C05488=1204.604,-6.269,-42.765,-179.791,5.566,148.916
C05489=1204.600,-6.020,-42.779,-179.789,5.567,148.915
C05490=1204.595,-5.770,-42.793,-179.786,5.567,148.915
C05491=1204.589,-5.521,-42.806,-179.783,5.568,148.914
C05492=1204.584,-5.271,-42.821,-179.781,5.568,148.913
C05493=1204.580,-5.022,-42.834,-179.779,5.568,148.913
C05494=1204.574,-4.772,-42.848,-179.776,5.569,148.912
C05495=1204.569,-4.522,-42.862,-179.773,5.569,148.911
C05496=1204.564,-4.273,-42.876,-179.771,5.570,148.911
C05497=1204.560,-4.024,-42.889,-179.769,5.570,148.910
C05498=1204.554,-3.774,-42.903,-179.766,5.571,148.909
C05499=1204.549,-3.525,-42.917,-179.764,5.571,148.909
C05500=1204.544,-3.275,-42.931,-179.761,5.571,148.908
C05501=1204.539,-3.025,-42.946,-179.759,5.572,148.907
C05502=1204.535,-2.776,-42.959,-179.756,5.572,148.907
C05503=1204.529,-2.526,-42.972,-179.754,5.573,148.906
C05504=1204.524,-2.276,-42.987,-179.751,5.573,148.905
C05505=1204.519,-2.027,-43.001,-179.749,5.573,148.905
C05506=1204.513,-1.778,-43.015,-179.746,5.574,148.904
C05507=1204.508,-1.528,-43.029,-179.744,5.574,148.903
C05508=1204.504,-1.278,-43.042,-179.741,5.575,148.903
C05509=1204.498,-1.029,-43.056,-179.738,5.575,148.902
C05510=1204.493,-0.779,-43.070,-179.736,5.576,148.902
C05511=1204.488,-0.529,-43.085,-179.734,5.576,148.901
C05512=1204.483,-0.280,-43.099,-179.732,5.576,148.900
C05513=1204.478,-0.031,-43.113,-179.729,5.577,148.899
C05514=1204.473,0.219,-43.127,-179.726,5.577,148.899
C05515=1204.468,0.469,-43.140,-179.724,5.578,148.898
C05516=1204.463,0.718,-43.154,-179.721,5.578,148.898
C05517=1204.458,0.968,-43.168,-179.719,5.579,148.897
C05518=1204.453,1.217,-43.182,-179.716,5.579,148.896
C05519=1204.448,1.467,-43.197,-179.714,5.579,148.896
C05520=1204.442,1.716,-43.211,-179.711,5.580,148.895
C05521=1204.437,1.966,-43.225,-179.709,5.580,148.894
C05522=1204.433,2.216,-43.239,-179.706,5.581,148.894
C05523=1204.428,2.465,-43.253,-179.704,5.582,148.893
C05524=1204.422,2.735,-43.268,-179.701,5.582,148.892
C05525=1204.416,3.003,-43.284,-179.698,5.582,148.891
C05526=1204.411,3.272,-43.299,-179.695,5.583,148.891
C05527=1204.406,3.542,-43.314,-179.693,5.583,148.890
C05528=1204.401,3.791,-43.328,-179.690,5.584,148.889
C05529=1204.396,4.041,-43.342,-179.688,5.585,148.889
C05530=1204.390,4.290,-43.356,-179.686,5.584,148.888
C05531=1204.385,4.540,-43.371,-179.683,5.585,148.888
C05532=1204.380,4.789,-43.385,-179.681,5.585,148.887
C05533=1204.376,5.039,-43.400,-179.678,5.586,148.886
C05534=1204.371,5.288,-43.414,-179.675,5.586,148.886
C05535=1204.365,5.537,-43.428,-179.673,5.587,148.885
C05536=1204.360,5.787,-43.442,-179.670,5.588,148.884
C05537=1204.355,6.037,-43.457,-179.668,5.588,148.884
C05538=1204.350,6.286,-43.471,-179.666,5.588,148.883
C05539=1204.345,6.536,-43.485,-179.663,5.588,148.882
C05540=1204.340,6.786,-43.499,-179.660,5.589,148.882
C05541=1204.335,7.035,-43.513,-179.658,5.589,148.881
C05542=1204.330,7.285,-43.528,-179.656,5.590,148.880
C05543=1204.325,7.534,-43.542,-179.653,5.591,148.880
C05544=1204.320,7.784,-43.556,-179.650,5.591,148.879
C05545=1204.315,8.033,-43.571,-179.648,5.592,148.878
C05546=1204.310,8.283,-43.585,-179.645,5.592,148.878
C05547=1204.305,8.532,-43.599,-179.643,5.592,148.877
C05548=1204.300,8.781,-43.614,-179.641,5.593,148.877
C05549=1204.295,9.031,-43.628,-179.638,5.593,148.876
C05550=1204.290,9.281,-43.642,-179.635,5.594,148.875
C05551=1204.285,9.530,-43.657,-179.633,5.594,148.875
C05552=1204.279,9.780,-43.672,-179.630,5.595,148.874
C05553=1204.275,10.030,-43.686,-179.628,5.595,148.873
C05554=1204.270,10.279,-43.701,-179.625,5.596,148.872
C05555=1204.264,10.528,-43.714,-179.623,5.597,148.872
C05556=1204.259,10.778,-43.729,-179.620,5.597,148.871
C05557=1204.254,11.027,-43.744,-179.618,5.597,148.871
C05558=1204.249,11.277,-43.758,-179.615,5.597,148.870
C05559=1204.244,11.527,-43.772,-179.613,5.598,148.869
C05560=1204.239,11.776,-43.788,-179.610,5.598,148.869
C05561=1204.234,12.026,-43.802,-179.608,5.599,148.868
C05562=1204.229,12.275,-43.816,-179.605,5.600,148.867
C05563=1204.224,12.525,-43.831,-179.603,5.600,148.867
C05564=1204.219,12.774,-43.845,-179.600,5.601,148.866
C05565=1204.214,13.023,-43.860,-179.597,5.601,148.865
C05566=1204.209,13.273,-43.874,-179.595,5.602,148.865
C05567=1204.204,13.522,-43.889,-179.593,5.602,148.864
C05568=1204.199,13.772,-43.904,-179.590,5.602,148.864
C05569=1204.194,14.022,-43.918,-179.588,5.603,148.863
C05570=1204.189,14.271,-43.933,-179.585,5.603,148.862
C05571=1204.184,14.521,-43.947,-179.582,5.604,148.862
C05572=1204.178,14.771,-43.962,-179.580,5.604,148.861
C05573=1204.174,15.020,-43.977,-179.578,5.605,148.860
C05574=1204.169,15.269,-43.991,-179.575,5.606,148.860
C05575=1204.164,15.519,-44.006,-179.572,5.606,148.859
C05576=1204.159,15.769,-44.021,-179.570,5.607,148.858
C05577=1204.154,16.018,-44.036,-179.567,5.607,148.858
C05578=1204.149,16.267,-44.051,-179.565,5.608,148.857
C05579=1204.144,16.517,-44.065,-179.562,5.609,148.857
C05580=1204.138,16.767,-44.080,-179.560,5.608,148.856
C05581=1204.134,17.016,-44.095,-179.558,5.609,148.855
C05582=1204.129,17.266,-44.109,-179.555,5.609,148.854
C05583=1204.124,17.515,-44.124,-179.552,5.610,148.854
C05584=1204.118,17.765,-44.139,-179.550,5.611,148.853
C05585=1204.114,18.014,-44.154,-179.547,5.611,148.853
C05586=1204.109,18.264,-44.168,-179.545,5.612,148.852
C05587=1204.104,18.514,-44.182,-179.542,5.612,148.851
C05588=1204.098,18.763,-44.198,-179.539,5.613,148.851
C05589=1204.093,19.013,-44.212,-179.537,5.613,148.850
C05590=1204.089,19.262,-44.227,-179.535,5.614,148.849
C05591=1204.083,19.512,-44.242,-179.532,5.615,148.849
C05592=1204.078,19.761,-44.257,-179.529,5.615,148.848
C05593=1204.074,20.010,-44.272,-179.527,5.616,148.847
C05594=1204.068,20.260,-44.287,-179.524,5.616,148.847
C05595=1204.063,20.509,-44.302,-179.522,5.617,148.846
C05596=1204.059,20.759,-44.316,-179.520,5.617,148.846
C05597=1204.053,21.008,-44.332,-179.517,5.617,148.845
C05598=1204.048,21.258,-44.346,-179.515,5.618,148.844
C05599=1204.044,21.507,-44.361,-179.512,5.618,148.844
C05600=1204.038,21.757,-44.376,-179.509,5.619,148.843
C05601=1204.033,22.006,-44.391,-179.507,5.620,148.842
C05602=1204.028,22.255,-44.407,-179.504,5.620,148.842
C05603=1204.023,22.505,-44.421,-179.502,5.621,148.841
C05604=1204.018,22.754,-44.436,-179.499,5.621,148.840
C05605=1204.012,23.004,-44.451,-179.497,5.622,148.840
C05606=1204.008,23.253,-44.466,-179.494,5.623,148.839
C05607=1204.002,23.503,-44.481,-179.492,5.623,148.839
C05608=1203.998,23.753,-44.496,-179.489,5.624,148.838
C05609=1203.993,24.002,-44.511,-179.486,5.624,148.837
C05610=1203.988,24.252,-44.527,-179.484,5.625,148.837
C05611=1203.983,24.501,-44.541,-179.482,5.626,148.836
C05612=1203.978,24.751,-44.556,-179.479,5.626,148.835
C05613=1203.973,25.000,-44.571,-179.476,5.627,148.835
C05614=1203.967,25.250,-44.586,-179.474,5.627,148.834
C05615=1203.963,25.499,-44.601,-179.471,5.628,148.833
C05616=1203.957,25.748,-44.617,-179.468,5.628,148.833
C05617=1203.953,25.998,-44.632,-179.466,5.629,148.832
C05618=1203.948,26.248,-44.646,-179.464,5.630,148.832
C05619=1203.943,26.497,-44.662,-179.461,5.630,148.831
C05620=1203.938,26.746,-44.677,-179.458,5.631,148.830
C05621=1203.933,26.996,-44.693,-179.456,5.631,148.830
C05622=1203.928,27.246,-44.707,-179.453,5.632,148.829
C05623=1203.923,27.495,-44.723,-179.451,5.632,148.828
C05624=1203.918,27.744,-44.738,-179.449,5.632,148.828
C05625=1203.913,27.994,-44.753,-179.446,5.633,148.827
C05626=1203.907,28.244,-44.768,-179.443,5.633,148.826
C05627=1203.903,28.493,-44.783,-179.441,5.634,148.826
C05628=1203.897,28.762,-44.800,-179.438,5.636,148.825
C05629=1203.892,29.030,-44.816,-179.435,5.636,148.825
C05630=1203.887,29.299,-44.833,-179.433,5.637,148.824
C05631=1203.881,29.568,-44.849,-179.430,5.637,148.823
C05632=1203.876,29.817,-44.864,-179.428,5.638,148.823
C05633=1203.871,30.067,-44.880,-179.425,5.638,148.822
C05634=1203.867,30.316,-44.895,-179.422,5.639,148.821
C05635=1203.861,30.566,-44.911,-179.420,5.639,148.820
C05636=1203.856,30.815,-44.925,-179.417,5.640,148.820
C05637=1203.851,31.065,-44.941,-179.415,5.641,148.819
C05638=1203.846,31.314,-44.956,-179.412,5.641,148.819
C05639=1203.841,31.564,-44.972,-179.410,5.642,148.818
C05640=1203.836,31.813,-44.987,-179.407,5.642,148.817
C05641=1203.831,32.063,-45.002,-179.405,5.643,148.817
C05642=1203.826,32.312,-45.018,-179.402,5.644,148.816
C05643=1203.821,32.562,-45.034,-179.399,5.644,148.816
C05644=1203.817,32.811,-45.049,-179.397,5.645,148.815
C05645=1203.811,33.061,-45.064,-179.395,5.646,148.814
C05646=1203.807,33.310,-45.079,-179.392,5.646,148.814
C05647=1203.801,33.559,-45.095,-179.389,5.647,148.813
C05648=1203.796,33.809,-45.111,-179.387,5.647,148.812
C05649=1203.792,34.058,-45.126,-179.384,5.648,148.812
C05650=1203.786,34.308,-45.142,-179.382,5.649,148.811
C05651=1203.781,34.557,-45.157,-179.379,5.649,148.811
C05652=1203.777,34.807,-45.172,-179.377,5.650,148.810
C05653=1203.772,35.056,-45.188,-179.374,5.650,148.809
C05654=1203.766,35.306,-45.204,-179.371,5.651,148.809
C05655=1203.761,35.555,-45.219,-179.369,5.652,148.808
C05656=1203.757,35.805,-45.235,-179.367,5.652,148.807
C05657=1203.751,36.054,-45.250,-179.364,5.653,148.807
C05658=1203.746,36.304,-45.266,-179.361,5.653,148.806
C05659=1203.742,36.553,-45.281,-179.359,5.654,148.806
C05660=1203.736,36.803,-45.297,-179.356,5.655,148.805
C05661=1203.731,37.052,-45.312,-179.354,5.655,148.804
C05662=1203.726,37.302,-45.328,-179.351,5.656,148.804
C05663=1203.722,37.551,-45.344,-179.349,5.656,148.803
C05664=1203.717,37.800,-45.360,-179.346,5.657,148.802
C05665=1203.711,38.050,-45.375,-179.344,5.658,148.802
C05666=1203.706,38.300,-45.391,-179.341,5.658,148.801
C05667=1203.702,38.549,-45.406,-179.338,5.659,148.800
C05668=1203.696,38.798,-45.422,-179.336,5.660,148.800
C05669=1203.692,39.048,-45.438,-179.334,5.660,148.799
C05670=1203.687,39.297,-45.454,-179.330,5.661,148.799
C05671=1203.681,39.547,-45.470,-179.328,5.662,148.798
C05672=1203.677,39.796,-45.485,-179.325,5.663,148.797
C05673=1203.672,40.046,-45.500,-179.323,5.663,148.797
C05674=1203.666,40.295,-45.516,-179.320,5.664,148.796
C05675=1203.662,40.545,-45.533,-179.318,5.664,148.796
C05676=1203.656,40.794,-45.548,-179.315,5.665,148.795
C05677=1203.652,41.043,-45.563,-179.313,5.666,148.794
C05678=1203.647,41.293,-45.579,-179.310,5.666,148.794
C05679=1203.642,41.543,-45.595,-179.308,5.667,148.793
C05680=1203.637,41.791,-45.611,-179.305,5.668,148.792
C05681=1203.632,42.041,-45.627,-179.303,5.668,148.792
C05682=1203.626,42.291,-45.643,-179.300,5.669,148.791
C05683=1203.621,42.540,-45.659,-179.298,5.669,148.791
C05684=1203.617,42.789,-45.674,-179.295,5.670,148.790
C05685=1203.612,43.039,-45.690,-179.293,5.671,148.789
C05686=1203.607,43.289,-45.706,-179.290,5.671,148.789
C05687=1203.602,43.538,-45.722,-179.288,5.672,148.788
C05688=1203.597,43.787,-45.738,-179.285,5.673,148.787
C05689=1203.592,44.037,-45.754,-179.283,5.673,148.787
C05690=1203.587,44.286,-45.770,-179.280,5.675,148.786
C05691=1203.582,44.536,-45.786,-179.277,5.675,148.786
C05692=1203.577,44.786,-45.802,-179.274,5.676,148.785
C05693=1203.572,45.034,-45.817,-179.272,5.677,148.785
C05694=1203.567,45.284,-45.833,-179.269,5.677,148.784
C05695=1203.562,45.533,-45.850,-179.267,5.678,148.783
C05696=1203.558,45.783,-45.866,-179.264,5.678,148.783
C05697=1203.552,46.032,-45.881,-179.262,5.679,148.782
C05698=1203.548,46.282,-45.898,-179.259,5.680,148.781
C05699=1203.542,46.531,-45.913,-179.257,5.680,148.781
C05700=1203.537,46.780,-45.930,-179.254,5.681,148.780
C05701=1203.532,47.030,-45.946,-179.252,5.682,148.780
C05702=1203.527,47.279,-45.962,-179.249,5.682,148.779
C05703=1203.523,47.529,-45.978,-179.246,5.684,148.778
C05704=1203.517,47.778,-45.993,-179.243,5.684,148.778
C05705=1203.513,48.028,-46.010,-179.241,5.685,148.777
C05706=1203.507,48.277,-46.026,-179.239,5.686,148.777
C05707=1203.503,48.527,-46.042,-179.236,5.686,148.776
C05708=1203.497,48.776,-46.058,-179.233,5.687,148.775
C05709=1203.493,49.026,-46.075,-179.231,5.688,148.775
C05710=1203.488,49.275,-46.090,-179.229,5.688,148.774
C05711=1203.483,49.525,-46.107,-179.226,5.689,148.773
C05712=1203.478,49.773,-46.123,-179.223,5.689,148.773
C05713=1203.473,50.024,-46.139,-179.221,5.690,148.772
C05714=1203.468,50.272,-46.155,-179.219,5.691,148.772
C05715=1203.463,50.522,-46.171,-179.215,5.692,148.771
C05716=1203.458,50.771,-46.188,-179.213,5.693,148.770
C05717=1203.454,51.021,-46.204,-179.211,5.693,148.770
C05718=1203.448,51.270,-46.220,-179.208,5.694,148.769
C05719=1203.443,51.520,-46.237,-179.205,5.694,148.769
C05720=1203.438,51.769,-46.253,-179.203,5.695,148.768
C05721=1203.433,52.019,-46.269,-179.200,5.696,148.767
C05722=1203.428,52.268,-46.285,-179.198,5.696,148.767
C05723=1203.423,52.518,-46.302,-179.195,5.697,148.766
C05724=1203.418,52.766,-46.318,-179.193,5.698,148.766
C05725=1203.414,53.017,-46.334,-179.190,5.699,148.765
C05726=1203.409,53.265,-46.350,-179.187,5.700,148.764
C05727=1203.404,53.515,-46.367,-179.185,5.700,148.764
C05728=1203.399,53.764,-46.383,-179.182,5.701,148.763
C05729=1203.393,54.014,-46.400,-179.180,5.702,148.763
C05730=1203.389,54.263,-46.417,-179.177,5.702,148.762
C05731=1203.384,54.513,-46.432,-179.175,5.703,148.761
C05732=1203.379,54.781,-46.450,-179.172,5.705,148.761
C05733=1203.373,55.050,-46.467,-179.169,5.705,148.760
C05734=1203.367,55.318,-46.486,-179.167,5.706,148.759
C05735=1203.362,55.587,-46.503,-179.164,5.706,148.759
C05736=1203.357,55.836,-46.519,-179.161,5.708,148.758
C05737=1203.353,56.086,-46.536,-179.158,5.708,148.757
C05738=1203.348,56.334,-46.552,-179.156,5.709,148.757
C05739=1203.342,56.585,-46.569,-179.153,5.710,148.756
C05740=1203.338,56.834,-46.585,-179.151,5.710,148.756
C05741=1203.333,57.083,-46.602,-179.148,5.711,148.755
C05742=1203.328,57.332,-46.618,-179.146,5.712,148.755
C05743=1203.322,57.582,-46.635,-179.143,5.712,148.754
C05744=1203.318,57.832,-46.651,-179.140,5.713,148.753
C05745=1203.313,58.081,-46.668,-179.138,5.714,148.753
C05746=1203.308,58.330,-46.684,-179.135,5.715,148.752
C05747=1203.304,58.579,-46.701,-179.133,5.715,148.751
C05748=1203.298,58.829,-46.718,-179.130,5.716,148.751
C05749=1203.293,59.078,-46.734,-179.128,5.717,148.750
C05750=1203.289,59.327,-46.751,-179.125,5.717,148.750
C05751=1203.283,59.577,-46.767,-179.122,5.719,148.749
C05752=1203.278,59.827,-46.784,-179.120,5.720,148.749
C05753=1203.274,60.076,-46.801,-179.117,5.720,148.748
C05754=1203.269,60.325,-46.817,-179.115,5.721,148.747
C05755=1203.263,60.575,-46.834,-179.112,5.722,148.747
C05756=1203.259,60.824,-46.851,-179.110,5.722,148.746
C05757=1203.254,61.073,-46.867,-179.107,5.723,148.746
C05758=1203.249,61.323,-46.884,-179.104,5.725,148.745
C05759=1203.244,61.572,-46.901,-179.102,5.725,148.744
C05760=1203.239,61.821,-46.917,-179.099,5.726,148.744
C05761=1203.234,62.071,-46.935,-179.097,5.726,148.743
C05762=1203.229,62.320,-46.951,-179.094,5.727,148.743
C05763=1203.225,62.570,-46.968,-179.092,5.728,148.742
C05764=1203.219,62.819,-46.985,-179.089,5.729,148.741
C05765=1203.215,63.068,-47.002,-179.086,5.730,148.741
C05766=1203.210,63.318,-47.018,-179.084,5.730,148.740
C05767=1203.204,63.567,-47.035,-179.081,5.731,148.740
C05768=1203.200,63.816,-47.052,-179.079,5.732,148.739
C05769=1203.195,64.066,-47.069,-179.076,5.732,148.738
C05770=1203.190,64.316,-47.086,-179.073,5.734,148.738
C05771=1203.185,64.565,-47.102,-179.071,5.735,148.737
C05772=1203.180,64.814,-47.119,-179.068,5.735,148.737
C05773=1203.175,65.064,-47.136,-179.066,5.736,148.736
C05774=1203.170,65.313,-47.153,-179.064,5.737,148.736
C05775=1203.165,65.562,-47.170,-179.061,5.737,148.735
C05776=1203.161,65.812,-47.186,-179.058,5.739,148.734
C05777=1203.155,66.062,-47.203,-179.056,5.740,148.734
C05778=1203.150,66.310,-47.220,-179.053,5.740,148.733
C05779=1203.145,66.560,-47.238,-179.050,5.741,148.733
C05780=1203.141,66.809,-47.254,-179.048,5.741,148.732
C05781=1203.136,67.059,-47.272,-179.045,5.743,148.731
C05782=1203.131,67.308,-47.288,-179.042,5.744,148.731
C05783=1203.125,67.557,-47.305,-179.040,5.744,148.730
C05784=1203.121,67.807,-47.322,-179.038,5.745,148.730
C05785=1203.116,68.057,-47.339,-179.035,5.746,148.729
C05786=1203.111,68.306,-47.357,-179.032,5.746,148.728
C05787=1203.106,68.555,-47.373,-179.030,5.748,148.728
C05788=1203.101,68.804,-47.390,-179.027,5.748,148.727
C05789=1203.096,69.054,-47.407,-179.024,5.749,148.727
C05790=1203.092,69.303,-47.425,-179.022,5.750,148.726
C05791=1203.087,69.553,-47.442,-179.020,5.750,148.726
C05792=1203.081,69.801,-47.458,-179.016,5.752,148.725
C05793=1203.076,70.051,-47.476,-179.014,5.753,148.724
C05794=1203.072,70.300,-47.493,-179.012,5.753,148.724
C05795=1203.067,70.550,-47.510,-179.009,5.754,148.723
C05796=1203.062,70.799,-47.527,-179.007,5.755,148.723
C05797=1203.057,71.049,-47.544,-179.004,5.756,148.722
C05798=1203.052,71.297,-47.561,-179.001,5.757,148.721
C05799=1203.047,71.547,-47.579,-178.999,5.758,148.721
C05800=1203.042,71.797,-47.596,-178.996,5.758,148.720
C05801=1203.038,72.046,-47.613,-178.994,5.760,148.720
C05802=1203.033,72.296,-47.630,-178.991,5.760,148.719
C05803=1203.028,72.545,-47.647,-178.988,5.761,148.719
C05804=1203.023,72.794,-47.665,-178.986,5.762,148.718
C05805=1203.017,73.043,-47.682,-178.984,5.762,148.717
C05806=1203.013,73.293,-47.699,-178.980,5.764,148.717
C05807=1203.008,73.542,-47.717,-178.978,5.765,148.716
C05808=1203.003,73.791,-47.733,-178.976,5.765,148.716
C05809=1202.998,74.041,-47.751,-178.973,5.766,148.715
C05810=1202.993,74.290,-47.769,-178.971,5.767,148.715
C05811=1202.989,74.540,-47.785,-178.968,5.768,148.714
C05812=1202.984,74.789,-47.803,-178.965,5.769,148.713
C05813=1202.978,75.038,-47.820,-178.963,5.770,148.713
C05814=1202.974,75.287,-47.837,-178.960,5.770,148.712
C05815=1202.969,75.537,-47.855,-178.957,5.772,148.712
C05816=1202.964,75.786,-47.873,-178.955,5.772,148.711
C05817=1202.959,76.036,-47.889,-178.952,5.773,148.710
C05818=1202.954,76.285,-47.907,-178.950,5.774,148.710
C05819=1202.949,76.535,-47.925,-178.947,5.775,148.709
C05820=1202.944,76.784,-47.942,-178.944,5.776,148.709
C05821=1202.940,77.033,-47.959,-178.942,5.777,148.708
C05822=1202.935,77.283,-47.977,-178.939,5.777,148.708
C05823=1202.930,77.532,-47.995,-178.936,5.779,148.707
C05824=1202.925,77.782,-48.011,-178.934,5.780,148.707
C05825=1202.920,78.031,-48.029,-178.931,5.780,148.706
C05826=1202.915,78.279,-48.047,-178.929,5.781,148.705
C05827=1202.910,78.529,-48.064,-178.926,5.783,148.705
C05828=1202.905,78.778,-48.081,-178.924,5.783,148.704
C05829=1202.900,79.028,-48.099,-178.921,5.784,148.704
C05830=1202.895,79.277,-48.117,-178.919,5.785,148.703
C05831=1202.890,79.527,-48.134,-178.916,5.786,148.702
C05832=1202.885,79.776,-48.152,-178.913,5.787,148.702
C05833=1202.881,80.025,-48.169,-178.911,5.787,148.701
C05834=1202.876,80.275,-48.187,-178.909,5.788,148.701
C05835=1202.871,80.524,-48.205,-178.905,5.790,148.700
C05836=1202.865,80.793,-48.223,-178.903,5.790,148.700
C05837=1202.860,81.061,-48.243,-178.900,5.791,148.699
C05838=1202.855,81.329,-48.262,-178.897,5.792,148.698
C05839=1202.849,81.597,-48.280,-178.895,5.793,148.698
C05840=1202.845,81.846,-48.298,-178.892,5.795,148.697
C05841=1202.840,82.096,-48.315,-178.889,5.795,148.697
C05842=1202.836,82.346,-48.333,-178.887,5.796,148.696
C05843=1202.831,82.595,-48.351,-178.884,5.797,148.696
C05844=1202.826,82.844,-48.369,-178.882,5.798,148.695
C05845=1202.821,83.094,-48.387,-178.879,5.799,148.694
C05846=1202.816,83.343,-48.405,-178.876,5.799,148.694
C05847=1202.811,83.592,-48.422,-178.874,5.801,148.693
C05848=1202.807,83.841,-48.440,-178.871,5.802,148.693
C05849=1202.801,84.091,-48.457,-178.869,5.803,148.692
C05850=1202.796,84.340,-48.475,-178.866,5.803,148.692
C05851=1202.792,84.589,-48.493,-178.863,5.805,148.691
C05852=1202.787,84.838,-48.511,-178.861,5.806,148.691
C05853=1202.781,85.088,-48.528,-178.858,5.806,148.690
C05854=1202.776,85.337,-48.546,-178.856,5.807,148.690
C05855=1202.772,85.587,-48.564,-178.853,5.808,148.689
C05856=1202.767,85.836,-48.582,-178.850,5.809,148.688
C05857=1202.762,86.085,-48.600,-178.848,5.810,148.688
C05858=1202.757,86.334,-48.618,-178.845,5.811,148.687
C05859=1202.752,86.584,-48.635,-178.843,5.812,148.687
C05860=1202.748,86.834,-48.653,-178.840,5.813,148.686
C05861=1202.743,87.083,-48.671,-178.837,5.814,148.685
C05862=1202.738,87.332,-48.689,-178.835,5.815,148.685
C05863=1202.733,87.581,-48.707,-178.832,5.816,148.684
C05864=1202.728,87.830,-48.725,-178.830,5.817,148.684
C05865=1202.723,88.079,-48.743,-178.827,5.818,148.683
C05866=1202.719,88.329,-48.761,-178.824,5.819,148.683
C05867=1202.714,88.578,-48.779,-178.822,5.820,148.682
C05868=1202.709,88.827,-48.797,-178.819,5.821,148.682
C05869=1202.704,89.076,-48.815,-178.817,5.822,148.681
C05870=1202.699,89.327,-48.833,-178.814,5.822,148.680
C05871=1202.694,89.576,-48.851,-178.812,5.824,148.680
C05872=1202.689,89.825,-48.869,-178.809,5.825,148.679
C05873=1202.684,90.074,-48.887,-178.806,5.825,148.679
C05874=1202.679,90.324,-48.905,-178.804,5.827,148.678
C05875=1202.674,90.573,-48.923,-178.801,5.828,148.678
C05876=1202.669,90.822,-48.941,-178.799,5.829,148.677
C05877=1202.665,91.072,-48.960,-178.796,5.830,148.677
C05878=1202.660,91.321,-48.978,-178.793,5.831,148.676
C05879=1202.655,91.570,-48.996,-178.791,5.831,148.676
C05880=1202.650,91.819,-49.014,-178.788,5.833,148.675
C05881=1202.645,92.068,-49.032,-178.786,5.834,148.675
C05882=1202.641,92.318,-49.051,-178.783,5.834,148.674
C05883=1202.636,92.567,-49.069,-178.781,5.835,148.673
C05884=1202.631,92.816,-49.087,-178.778,5.837,148.673
C05885=1202.626,93.066,-49.105,-178.775,5.838,148.672
C05886=1202.621,93.315,-49.123,-178.773,5.838,148.672
C05887=1202.616,93.565,-49.141,-178.770,5.840,148.671
C05888=1202.611,93.814,-49.159,-178.768,5.840,148.671
C05889=1202.607,94.063,-49.177,-178.764,5.842,148.670
C05890=1202.602,94.312,-49.196,-178.762,5.843,148.670
C05891=1202.597,94.561,-49.214,-178.760,5.843,148.669
C05892=1202.592,94.811,-49.233,-178.757,5.845,148.669
C05893=1202.587,95.060,-49.251,-178.754,5.846,148.668
C05894=1202.582,95.309,-49.269,-178.752,5.847,148.667
C05895=1202.577,95.558,-49.287,-178.749,5.848,148.667
C05896=1202.573,95.807,-49.306,-178.747,5.849,148.666
C05897=1202.568,96.057,-49.325,-178.744,5.850,148.666
C05898=1202.563,96.306,-49.343,-178.741,5.851,148.665
C05899=1202.558,96.556,-49.361,-178.739,5.852,148.665
C05900=1202.553,96.805,-49.379,-178.736,5.852,148.664
C05901=1202.549,97.054,-49.398,-178.734,5.854,148.664
C05902=1202.543,97.304,-49.416,-178.731,5.855,148.663
C05903=1202.538,97.553,-49.434,-178.729,5.856,148.663
C05904=1202.534,97.802,-49.453,-178.726,5.857,148.662
C05905=1202.529,98.051,-49.471,-178.723,5.858,148.662
C05906=1202.524,98.301,-49.490,-178.721,5.859,148.661
C05907=1202.519,98.550,-49.508,-178.718,5.860,148.660
C05908=1202.515,98.799,-49.527,-178.716,5.861,148.660
C05909=1202.510,99.048,-49.545,-178.713,5.863,148.659
C05910=1202.504,99.298,-49.563,-178.710,5.863,148.659
C05911=1202.500,99.547,-49.582,-178.708,5.864,148.658
C05912=1202.495,99.796,-49.600,-178.705,5.866,148.658
C05913=1202.490,100.046,-49.619,-178.702,5.866,148.657
C05914=1202.486,100.295,-49.638,-178.700,5.867,148.657
C05915=1202.481,100.544,-49.656,-178.697,5.868,148.656
C05916=1202.475,100.793,-49.675,-178.695,5.869,148.656
C05917=1202.470,101.042,-49.693,-178.692,5.871,148.655
C05918=1202.466,101.292,-49.712,-178.689,5.872,148.655
C05919=1202.461,101.541,-49.731,-178.687,5.872,148.654
C05920=1202.456,101.790,-49.749,-178.684,5.874,148.653
C05921=1202.452,102.039,-49.768,-178.682,5.875,148.653
C05922=1202.446,102.289,-49.787,-178.679,5.876,148.652
C05923=1202.442,102.538,-49.806,-178.676,5.877,148.652
C05924=1202.437,102.787,-49.824,-178.674,5.878,148.651
C05925=1202.432,103.037,-49.842,-178.671,5.879,148.651
C05926=1202.428,103.286,-49.861,-178.669,5.880,148.650
C05927=1202.422,103.535,-49.880,-178.666,5.881,148.650
C05928=1202.417,103.784,-49.898,-178.663,5.883,148.649
C05929=1202.413,104.034,-49.917,-178.661,5.883,148.649
C05930=1202.408,104.283,-49.936,-178.658,5.885,148.648
C05931=1202.403,104.532,-49.954,-178.656,5.886,148.648
C05932=1202.398,104.781,-49.974,-178.653,5.886,148.647
C05933=1202.394,105.030,-49.992,-178.650,5.888,148.647
C05934=1202.388,105.280,-50.011,-178.648,5.889,148.646
C05935=1202.384,105.529,-50.030,-178.645,5.890,148.645
C05936=1202.379,105.778,-50.048,-178.643,5.891,148.645
C05937=1202.374,106.028,-50.068,-178.640,5.893,148.644
C05938=1202.369,106.277,-50.086,-178.637,5.893,148.644
C05939=1202.365,106.526,-50.105,-178.635,5.894,148.643
C05940=1202.359,106.794,-50.126,-178.632,5.895,148.643
C05941=1202.354,107.062,-50.145,-178.629,5.897,148.642
C05942=1202.349,107.331,-50.167,-178.626,5.898,148.642
C05943=1202.343,107.600,-50.187,-178.623,5.899,148.641
C05944=1202.339,107.849,-50.206,-178.621,5.900,148.641
C05945=1202.334,108.098,-50.224,-178.618,5.902,148.640
C05946=1202.330,108.348,-50.243,-178.616,5.903,148.640
C05947=1202.324,108.597,-50.263,-178.614,5.903,148.639
C05948=1202.320,108.846,-50.282,-178.610,5.905,148.639
C05949=1202.315,109.095,-50.300,-178.608,5.906,148.638
C05950=1202.310,109.344,-50.319,-178.605,5.907,148.638
C05951=1202.305,109.593,-50.339,-178.603,5.908,148.637
C05952=1202.300,109.843,-50.357,-178.600,5.910,148.636
C05953=1202.296,110.092,-50.376,-178.598,5.910,148.636
C05954=1202.290,110.341,-50.395,-178.594,5.912,148.635
C05955=1202.286,110.590,-50.415,-178.592,5.913,148.635
C05956=1202.281,110.840,-50.433,-178.590,5.913,148.634
C05957=1202.277,111.089,-50.452,-178.587,5.915,148.634
C05958=1202.271,111.338,-50.471,-178.584,5.916,148.633
C05959=1202.267,111.587,-50.491,-178.582,5.918,148.633
C05960=1202.262,111.836,-50.510,-178.579,5.918,148.632
C05961=1202.257,112.086,-50.529,-178.576,5.920,148.632
C05962=1202.252,112.335,-50.547,-178.574,5.920,148.631
C05963=1202.247,112.584,-50.567,-178.571,5.922,148.631
C05964=1202.242,112.833,-50.586,-178.569,5.923,148.630
C05965=1202.238,113.082,-50.605,-178.566,5.924,148.630
C05966=1202.233,113.332,-50.625,-178.564,5.926,148.629
C05967=1202.228,113.581,-50.644,-178.561,5.926,148.629
C05968=1202.224,113.831,-50.663,-178.558,5.928,148.628
C05969=1202.218,114.080,-50.682,-178.556,5.928,148.628
C05970=1202.214,114.329,-50.702,-178.553,5.930,148.627
C05971=1202.209,114.578,-50.720,-178.550,5.931,148.627
C05972=1202.204,114.827,-50.740,-178.548,5.933,148.626
C05973=1202.199,115.076,-50.759,-178.545,5.933,148.626
C05974=1202.195,115.325,-50.778,-178.542,5.935,148.625
C05975=1202.190,115.574,-50.798,-178.540,5.936,148.625
C05976=1202.185,115.824,-50.817,-178.537,5.937,148.624
C05977=1202.180,116.073,-50.837,-178.535,5.938,148.624
C05978=1202.175,116.322,-50.856,-178.532,5.939,148.623
C05979=1202.171,116.572,-50.875,-178.530,5.941,148.623
C05980=1202.165,116.820,-50.895,-178.527,5.941,148.622
C05981=1202.161,117.070,-50.914,-178.524,5.943,148.622
C05982=1202.157,117.319,-50.933,-178.522,5.944,148.621
C05983=1202.151,117.568,-50.953,-178.519,5.945,148.621
C05984=1202.147,117.818,-50.972,-178.517,5.946,148.620
C05985=1202.141,118.067,-50.992,-178.514,5.948,148.620
C05986=1202.136,118.316,-51.011,-178.512,5.949,148.619
C05987=1202.132,118.565,-51.030,-178.508,5.950,148.619
C05988=1202.127,118.814,-51.050,-178.506,5.951,148.618
C05989=1202.122,119.064,-51.069,-178.503,5.952,148.618
C05990=1202.118,119.313,-51.089,-178.501,5.953,148.617
C05991=1202.112,119.562,-51.108,-178.498,5.955,148.617
C05992=1202.109,119.811,-51.128,-178.496,5.956,148.616
C05993=1202.103,120.060,-51.147,-178.493,5.957,148.616
C05994=1202.099,120.309,-51.167,-178.490,5.958,148.615
C05995=1202.094,120.559,-51.187,-178.488,5.960,148.615
C05996=1202.088,120.808,-51.206,-178.486,5.961,148.614
C05997=1202.084,121.057,-51.226,-178.482,5.962,148.614
C05998=1202.079,121.306,-51.246,-178.480,5.963,148.613
C05999=1202.075,121.555,-51.265,-178.477,5.965,148.613
C06000=1202.070,121.804,-51.284,-178.475,5.965,148.612
C06001=1202.065,122.054,-51.304,-178.472,5.967,148.612
C06002=1202.060,122.304,-51.324,-178.470,5.968,148.611
C06003=1202.055,122.552,-51.344,-178.467,5.970,148.611
C06004=1202.051,122.801,-51.363,-178.464,5.970,148.610
C06005=1202.046,123.051,-51.383,-178.462,5.972,148.610
C06006=1202.041,123.300,-51.402,-178.459,5.973,148.609
C06007=1202.036,123.549,-51.423,-178.456,5.974,148.609
C06008=1202.031,123.798,-51.442,-178.454,5.975,148.608
C06009=1202.026,124.047,-51.462,-178.451,5.977,148.608
C06010=1202.022,124.296,-51.481,-178.449,5.978,148.607
C06011=1202.018,124.545,-51.501,-178.446,5.979,148.607
C06012=1202.013,124.795,-51.521,-178.444,5.980,148.606
C06013=1202.007,125.044,-51.540,-178.441,5.982,148.606
C06014=1202.003,125.293,-51.560,-178.438,5.983,148.605
C06015=1201.998,125.542,-51.580,-178.436,5.984,148.605
C06016=1201.994,125.792,-51.600,-178.433,5.986,148.604
C06017=1201.989,126.040,-51.620,-178.430,5.987,148.604
C06018=1201.984,126.290,-51.639,-178.428,5.988,148.603
C06019=1201.979,126.539,-51.660,-178.425,5.989,148.603
C06020=1201.975,126.788,-51.679,-178.422,5.991,148.602
C06021=1201.969,127.037,-51.699,-178.420,5.992,148.602
C06022=1201.965,127.286,-51.719,-178.417,5.993,148.601
C06023=1201.960,127.536,-51.739,-178.415,5.994,148.601
C06024=1201.956,127.785,-51.759,-178.412,5.995,148.600
C06025=1201.951,128.034,-51.779,-178.410,5.996,148.600
C06026=1201.946,128.282,-51.799,-178.407,5.998,148.600
C06027=1201.940,128.532,-51.819,-178.404,6.000,148.599
C06028=1201.936,128.782,-51.839,-178.402,6.001,148.599
C06029=1201.931,129.031,-51.859,-178.399,6.002,148.598
C06030=1201.926,129.280,-51.879,-178.396,6.003,148.598
C06031=1201.921,129.529,-51.899,-178.394,6.005,148.597
C06032=1201.917,129.778,-51.918,-178.391,6.005,148.596
C06033=1201.912,130.027,-51.939,-178.389,6.007,148.596
C06034=1201.908,130.276,-51.959,-178.386,6.008,148.596
C06035=1201.903,130.526,-51.979,-178.383,6.009,148.595
C06036=1201.899,130.775,-51.999,-178.381,6.011,148.595
C06037=1201.893,131.024,-52.019,-178.378,6.012,148.594
C06038=1201.888,131.273,-52.039,-178.375,6.014,148.594
C06039=1201.883,131.522,-52.059,-178.373,6.015,148.593
C06040=1201.879,131.771,-52.079,-178.370,6.016,148.593
C06041=1201.874,132.020,-52.100,-178.368,6.017,148.592
C06042=1201.870,132.270,-52.119,-178.365,6.019,148.592
C06043=1201.864,132.518,-52.140,-178.362,6.020,148.591
C06044=1201.860,132.788,-52.161,-178.360,6.021,148.591
C06045=1201.854,133.056,-52.184,-178.357,6.022,148.590
C06046=1201.849,133.325,-52.205,-178.354,6.024,148.590
C06047=1201.844,133.593,-52.227,-178.351,6.026,148.589
C06048=1201.839,133.843,-52.247,-178.349,6.027,148.589
C06049=1201.835,134.092,-52.267,-178.346,6.028,148.588
C06050=1201.830,134.340,-52.288,-178.343,6.029,148.588
C06051=1201.824,134.590,-52.308,-178.341,6.031,148.587
C06052=1201.820,134.839,-52.328,-178.338,6.033,148.587
C06053=1201.815,135.088,-52.348,-178.335,6.033,148.586
C06054=1201.811,135.337,-52.368,-178.333,6.035,148.586
C06055=1201.806,135.586,-52.389,-178.331,6.036,148.586
C06056=1201.801,135.835,-52.409,-178.327,6.037,148.585
C06057=1201.797,136.084,-52.430,-178.325,6.039,148.585
C06058=1201.792,136.334,-52.449,-178.323,6.040,148.584
C06059=1201.787,136.583,-52.470,-178.320,6.042,148.584
C06060=1201.782,136.832,-52.491,-178.317,6.042,148.583
C06061=1201.778,137.081,-52.511,-178.315,6.044,148.583
C06062=1201.773,137.330,-52.532,-178.312,6.046,148.582
C06063=1201.768,137.579,-52.552,-178.309,6.047,148.582
C06064=1201.764,137.829,-52.572,-178.307,6.048,148.581
C06065=1201.758,138.078,-52.593,-178.304,6.049,148.581
C06066=1201.753,138.326,-52.613,-178.301,6.051,148.580
C06067=1201.749,138.575,-52.633,-178.299,6.053,148.580
C06068=1201.744,138.824,-52.654,-178.297,6.054,148.580
C06069=1201.739,139.073,-52.675,-178.293,6.055,148.579
C06070=1201.735,139.322,-52.695,-178.291,6.057,148.579
C06071=1201.730,139.572,-52.716,-178.289,6.058,148.578
C06072=1201.725,139.821,-52.736,-178.286,6.059,148.578
C06073=1201.720,140.070,-52.756,-178.283,6.060,148.577
C06074=1201.715,140.319,-52.777,-178.281,6.062,148.577
C06075=1201.711,140.568,-52.797,-178.278,6.063,148.576
C06076=1201.706,140.818,-52.818,-178.275,6.064,148.576
C06077=1201.701,141.067,-52.839,-178.273,6.066,148.575
C06078=1201.697,141.316,-52.859,-178.270,6.068,148.575
C06079=1201.692,141.565,-52.880,-178.267,6.068,148.574
C06080=1201.687,141.814,-52.900,-178.265,6.070,148.574
C06081=1201.683,142.064,-52.922,-178.263,6.071,148.574
C06082=1201.678,142.313,-52.942,-178.260,6.073,148.573
C06083=1201.673,142.562,-52.963,-178.257,6.074,148.573
C06084=1201.669,142.811,-52.983,-178.255,6.075,148.572
C06085=1201.664,143.060,-53.004,-178.252,6.077,148.572
C06086=1201.659,143.309,-53.025,-178.249,6.079,148.571
C06087=1201.655,143.558,-53.045,-178.247,6.080,148.571
C06088=1201.649,143.807,-53.066,-178.244,6.081,148.570
C06089=1201.645,144.056,-53.087,-178.241,6.083,148.570
C06090=1201.640,144.305,-53.108,-178.239,6.084,148.569
C06091=1201.636,144.554,-53.129,-178.236,6.085,148.569
C06092=1201.630,144.803,-53.150,-178.233,6.087,148.569
C06093=1201.626,145.052,-53.170,-178.231,6.088,148.568
C06094=1201.621,145.301,-53.191,-178.228,6.090,148.568
C06095=1201.616,145.550,-53.211,-178.225,6.091,148.567
C06096=1201.612,145.800,-53.233,-178.223,6.092,148.567
C06097=1201.607,146.049,-53.254,-178.220,6.094,148.566
C06098=1201.603,146.298,-53.275,-178.218,6.096,148.566
C06099=1201.597,146.547,-53.296,-178.215,6.097,148.566
C06100=1201.593,146.796,-53.316,-178.212,6.098,148.565
C06101=1201.588,147.045,-53.337,-178.210,6.100,148.565
C06102=1201.584,147.294,-53.358,-178.207,6.101,148.564
C06103=1201.578,147.543,-53.379,-178.205,6.103,148.564
C06104=1201.574,147.793,-53.400,-178.202,6.104,148.563
C06105=1201.569,148.042,-53.421,-178.200,6.105,148.563
C06106=1201.565,148.290,-53.442,-178.197,6.107,148.562
C06107=1201.560,148.539,-53.463,-178.194,6.109,148.562
C06108=1201.555,148.789,-53.484,-178.192,6.109,148.561
C06109=1201.550,149.037,-53.505,-178.189,6.111,148.561
C06110=1201.546,149.286,-53.526,-178.186,6.113,148.561
C06111=1201.541,149.536,-53.547,-178.184,6.114,148.560
C06112=1201.536,149.785,-53.568,-178.181,6.115,148.560
C06113=1201.532,150.034,-53.589,-178.178,6.117,148.559
C06114=1201.527,150.283,-53.610,-178.176,6.118,148.559
C06115=1201.521,150.532,-53.631,-178.173,6.120,148.559
C06116=1201.517,150.781,-53.652,-178.170,6.121,148.558
C06117=1201.513,151.031,-53.674,-178.168,6.122,148.558
C06118=1201.508,151.279,-53.695,-178.166,6.124,148.557
C06119=1201.503,151.528,-53.716,-178.163,6.126,148.557
C06120=1201.498,151.777,-53.737,-178.160,6.127,148.556
C06121=1201.493,152.026,-53.758,-178.158,6.128,148.556
C06122=1201.489,152.276,-53.779,-178.155,6.130,148.555
C06123=1201.485,152.524,-53.801,-178.152,6.132,148.555
C06124=1201.479,152.774,-53.822,-178.150,6.132,148.554
C06125=1201.475,153.022,-53.843,-178.147,6.134,148.554
C06126=1201.471,153.272,-53.864,-178.144,6.136,148.554
C06127=1201.466,153.520,-53.886,-178.142,6.137,148.553
C06128=1201.461,153.770,-53.907,-178.139,6.139,148.553
C06129=1201.456,154.018,-53.928,-178.136,6.140,148.552
C06130=1201.451,154.267,-53.949,-178.134,6.142,148.552
C06131=1201.447,154.517,-53.971,-178.132,6.143,148.552
C06132=1201.442,154.766,-53.992,-178.129,6.145,148.551
C06133=1201.437,155.015,-54.013,-178.126,6.146,148.551
C06134=1201.432,155.264,-54.034,-178.124,6.147,148.550
C06135=1201.428,155.513,-54.056,-178.121,6.149,148.550
C06136=1201.423,155.762,-54.077,-178.118,6.151,148.549
C06137=1201.418,156.011,-54.099,-178.116,6.152,148.549
C06138=1201.414,156.261,-54.120,-178.113,6.153,148.548
C06139=1201.409,156.509,-54.142,-178.110,6.155,148.548
C06140=1201.404,156.758,-54.163,-178.108,6.157,148.548
C06141=1201.399,157.007,-54.184,-178.105,6.158,148.547
C06142=1201.395,157.256,-54.206,-178.103,6.159,148.547
C06143=1201.390,157.505,-54.227,-178.100,6.161,148.546
C06144=1201.385,157.754,-54.248,-178.097,6.163,148.546
C06145=1201.381,158.004,-54.270,-178.094,6.164,148.546
C06146=1201.376,158.252,-54.292,-178.092,6.165,148.545
C06147=1201.371,158.501,-54.313,-178.090,6.167,148.545
C06148=1201.367,158.770,-54.336,-178.086,6.169,148.544
C06149=1201.361,159.039,-54.360,-178.084,6.170,148.544
C06150=1201.356,159.308,-54.383,-178.081,6.172,148.543
C06151=1201.351,159.578,-54.406,-178.078,6.174,148.543
C06152=1201.347,159.827,-54.428,-178.075,6.175,148.542
C06153=1201.342,160.076,-54.450,-178.073,6.176,148.542
C06154=1201.337,160.324,-54.471,-178.070,6.178,148.542
C06155=1201.332,160.574,-54.493,-178.068,6.180,148.541
C06156=1201.327,160.823,-54.514,-178.065,6.181,148.541
C06157=1201.322,161.072,-54.536,-178.062,6.182,148.540
C06158=1201.318,161.321,-54.558,-178.060,6.184,148.540
C06159=1201.313,161.569,-54.580,-178.057,6.186,148.540
C06160=1201.308,161.819,-54.601,-178.054,6.188,148.539
C06161=1201.304,162.068,-54.623,-178.052,6.189,148.539
C06162=1201.299,162.317,-54.644,-178.049,6.190,148.538
C06163=1201.295,162.566,-54.667,-178.047,6.192,148.538
C06164=1201.290,162.815,-54.688,-178.044,6.194,148.538
C06165=1201.285,163.063,-54.710,-178.041,6.196,148.537
C06166=1201.281,163.313,-54.732,-178.039,6.196,148.537
C06167=1201.276,163.561,-54.754,-178.036,6.198,148.536
C06168=1201.271,163.811,-54.775,-178.033,6.200,148.536
C06169=1201.266,164.060,-54.797,-178.031,6.202,148.535
C06170=1201.262,164.309,-54.819,-178.028,6.203,148.535
C06171=1201.257,164.558,-54.840,-178.026,6.204,148.535
C06172=1201.252,164.807,-54.862,-178.023,6.206,148.534
C06173=1201.248,165.056,-54.884,-178.020,6.208,148.534
C06174=1201.243,165.305,-54.906,-178.018,6.210,148.534
C06175=1201.239,165.554,-54.928,-178.015,6.210,148.533
C06176=1201.234,165.803,-54.949,-178.013,6.212,148.533
C06177=1201.230,166.052,-54.972,-178.010,6.214,148.532
C06178=1201.225,166.300,-54.993,-178.007,6.216,148.532
C06179=1201.220,166.550,-55.016,-178.005,6.218,148.532
C06180=1201.215,166.799,-55.038,-178.002,6.218,148.531
C06181=1201.211,167.048,-55.060,-178.000,6.220,148.531
C06182=1201.206,167.297,-55.081,-177.997,6.222,148.530
C06183=1201.202,167.546,-55.103,-177.994,6.224,148.530
C06184=1201.197,167.795,-55.125,-177.991,6.225,148.529
C06185=1201.193,168.043,-55.148,-177.989,6.226,148.529
C06186=1201.187,168.292,-55.170,-177.987,6.228,148.529
C06187=1201.183,168.542,-55.192,-177.984,6.230,148.528
C06188=1201.178,168.790,-55.214,-177.981,6.232,148.528
C06189=1201.174,169.040,-55.236,-177.979,6.234,148.528
C06190=1201.169,169.288,-55.258,-177.976,6.234,148.527
C06191=1201.164,169.538,-55.280,-177.973,6.236,148.527
C06192=1201.159,169.787,-55.302,-177.971,6.238,148.526
C06193=1201.155,170.035,-55.325,-177.968,6.240,148.526
C06194=1201.150,170.284,-55.346,-177.965,6.241,148.526
C06195=1201.145,170.534,-55.369,-177.963,6.243,148.525
C06196=1201.140,170.782,-55.391,-177.960,6.244,148.525
C06197=1201.136,171.032,-55.413,-177.958,6.246,148.524
C06198=1201.132,171.280,-55.435,-177.955,6.247,148.524
C06199=1201.127,171.529,-55.458,-177.952,6.249,148.523
C06200=1201.122,171.778,-55.479,-177.949,6.251,148.523
C06201=1201.117,172.027,-55.501,-177.947,6.252,148.523
C06202=1201.113,172.276,-55.525,-177.945,6.254,148.522
C06203=1201.108,172.525,-55.546,-177.942,6.256,148.522
C06204=1201.104,172.774,-55.569,-177.939,6.257,148.522
C06205=1201.099,173.023,-55.590,-177.937,6.259,148.521
C06206=1201.094,173.272,-55.614,-177.934,6.261,148.521
C06207=1201.090,173.521,-55.636,-177.931,6.263,148.521
C06208=1201.085,173.770,-55.657,-177.929,6.264,148.520
C06209=1201.080,174.019,-55.681,-177.926,6.265,148.520
C06210=1201.075,174.268,-55.702,-177.923,6.267,148.519
C06211=1201.071,174.517,-55.724,-177.921,6.269,148.519
C06212=1201.066,174.766,-55.748,-177.918,6.271,148.518
C06213=1201.062,175.015,-55.769,-177.915,6.272,148.518
C06214=1201.057,175.264,-55.793,-177.913,6.273,148.518
C06215=1201.052,175.512,-55.814,-177.911,6.275,148.517
C06216=1201.048,175.762,-55.837,-177.908,6.277,148.517
C06217=1201.043,176.011,-55.860,-177.905,6.279,148.517
C06218=1201.038,176.259,-55.882,-177.903,6.281,148.516
C06219=1201.033,176.508,-55.905,-177.900,6.282,148.516
C06220=1201.029,176.758,-55.927,-177.897,6.284,148.516
C06221=1201.025,177.006,-55.949,-177.895,6.285,148.515
C06222=1201.020,177.255,-55.972,-177.892,6.287,148.515
C06223=1201.016,177.504,-55.995,-177.889,6.288,148.514
C06224=1201.010,177.753,-56.017,-177.887,6.290,148.514
C06225=1201.006,178.002,-56.040,-177.884,6.292,148.514
C06226=1201.001,178.251,-56.062,-177.881,6.294,148.513
C06227=1200.997,178.499,-56.085,-177.879,6.296,148.513
C06228=1200.991,178.749,-56.107,-177.876,6.297,148.512
C06229=1200.988,178.998,-56.130,-177.874,6.298,148.512
C06230=1200.982,179.247,-56.153,-177.871,6.300,148.512
C06231=1200.978,179.496,-56.175,-177.869,6.302,148.511
C06232=1200.973,179.745,-56.199,-177.866,6.304,148.511
C06233=1200.969,179.994,-56.221,-177.863,6.306,148.511
C06234=1200.964,180.242,-56.244,-177.861,6.307,148.510
C06235=1200.959,180.492,-56.266,-177.858,6.309,148.510
C06236=1200.955,180.741,-56.289,-177.855,6.311,148.510
C06237=1200.950,180.989,-56.312,-177.853,6.313,148.509
C06238=1200.945,181.238,-56.334,-177.850,6.314,148.509
C06239=1200.941,181.487,-56.357,-177.848,6.316,148.508
C06240=1200.936,181.736,-56.380,-177.845,6.317,148.508
C06241=1200.932,181.985,-56.402,-177.842,6.319,148.508
C06242=1200.927,182.234,-56.425,-177.839,6.321,148.507
C06243=1200.923,182.482,-56.448,-177.837,6.323,148.507
C06244=1200.918,182.732,-56.471,-177.834,6.324,148.506
C06245=1200.913,182.980,-56.494,-177.831,6.326,148.506
C06246=1200.909,183.229,-56.516,-177.829,6.328,148.506
C06247=1200.904,183.478,-56.540,-177.826,6.330,148.505
C06248=1200.900,183.728,-56.562,-177.823,6.332,148.505
C06249=1200.895,183.977,-56.585,-177.821,6.333,148.505
C06250=1200.890,184.225,-56.608,-177.819,6.334,148.504
C06251=1200.886,184.474,-56.631,-177.816,6.336,148.504
C06252=1200.880,184.743,-56.656,-177.813,6.338,148.504
C06253=1200.875,185.013,-56.681,-177.810,6.341,148.503
C06254=1200.871,185.283,-56.706,-177.807,6.342,148.503
C06255=1200.865,185.552,-56.731,-177.804,6.344,148.502
C06256=1200.861,185.801,-56.754,-177.802,6.346,148.502
C06257=1200.857,186.050,-56.777,-177.799,6.348,148.502
C06258=1200.852,186.299,-56.800,-177.796,6.349,148.501
C06259=1200.847,186.547,-56.823,-177.794,6.351,148.501
C06260=1200.842,186.797,-56.845,-177.791,6.353,148.501
C06261=1200.838,187.046,-56.868,-177.789,6.354,148.500
C06262=1200.833,187.295,-56.892,-177.786,6.356,148.500
C06263=1200.828,187.544,-56.915,-177.784,6.358,148.500
C06264=1200.824,187.793,-56.938,-177.781,6.359,148.499
C06265=1200.820,188.042,-56.961,-177.778,6.361,148.499
C06266=1200.814,188.290,-56.984,-177.776,6.363,148.498
C06267=1200.810,188.539,-57.008,-177.773,6.365,148.498
C06268=1200.806,188.788,-57.030,-177.770,6.367,148.498
C06269=1200.801,189.037,-57.054,-177.768,6.368,148.497
C06270=1200.796,189.286,-57.077,-177.765,6.370,148.497
C06271=1200.791,189.535,-57.100,-177.762,6.372,148.497
C06272=1200.788,189.784,-57.123,-177.760,6.374,148.496
C06273=1200.783,190.033,-57.147,-177.757,6.376,148.496
C06274=1200.778,190.281,-57.170,-177.755,6.378,148.496
C06275=1200.773,190.530,-57.193,-177.752,6.380,148.496
C06276=1200.768,190.779,-57.216,-177.750,6.381,148.495
C06277=1200.763,191.028,-57.240,-177.747,6.383,148.495
C06278=1200.759,191.277,-57.262,-177.744,6.385,148.494
C06279=1200.755,191.525,-57.286,-177.742,6.387,148.494
C06280=1200.750,191.774,-57.310,-177.739,6.389,148.494
C06281=1200.746,192.023,-57.333,-177.736,6.390,148.493
C06282=1200.741,192.272,-57.357,-177.734,6.391,148.493
C06283=1200.736,192.521,-57.380,-177.731,6.393,148.493
C06284=1200.732,192.770,-57.403,-177.729,6.395,148.492
C06285=1200.727,193.019,-57.427,-177.726,6.397,148.492
C06286=1200.723,193.267,-57.450,-177.723,6.399,148.492
C06287=1200.718,193.516,-57.473,-177.721,6.401,148.491
C06288=1200.714,193.766,-57.497,-177.718,6.402,148.491
C06289=1200.709,194.014,-57.520,-177.716,6.404,148.491
C06290=1200.704,194.263,-57.543,-177.713,6.406,148.490
C06291=1200.699,194.511,-57.567,-177.710,6.408,148.490
C06292=1200.695,194.760,-57.591,-177.708,6.410,148.490
C06293=1200.690,195.009,-57.614,-177.705,6.411,148.489
C06294=1200.685,195.258,-57.637,-177.702,6.413,148.489
C06295=1200.681,195.507,-57.661,-177.700,6.415,148.489
C06296=1200.676,195.756,-57.685,-177.697,6.417,148.488
C06297=1200.672,196.005,-57.708,-177.694,6.419,148.488
C06298=1200.667,196.253,-57.732,-177.692,6.421,148.488
C06299=1200.662,196.502,-57.756,-177.689,6.423,148.487
C06300=1200.658,196.751,-57.779,-177.687,6.424,148.487
C06301=1200.653,197.000,-57.803,-177.684,6.426,148.487
C06302=1200.649,197.249,-57.826,-177.681,6.428,148.486
C06303=1200.645,197.499,-57.850,-177.679,6.430,148.486
C06304=1200.640,197.747,-57.874,-177.676,6.432,148.486
C06305=1200.635,197.996,-57.898,-177.674,6.434,148.485
C06306=1200.631,198.245,-57.921,-177.671,6.435,148.485
C06307=1200.626,198.493,-57.945,-177.668,6.437,148.485
C06308=1200.622,198.742,-57.968,-177.666,6.439,148.484
C06309=1200.617,198.991,-57.992,-177.663,6.441,148.484
C06310=1200.613,199.240,-58.016,-177.660,6.443,148.484
C06311=1200.608,199.488,-58.040,-177.658,6.444,148.483
C06312=1200.603,199.738,-58.064,-177.655,6.447,148.483
C06313=1200.598,199.987,-58.087,-177.653,6.448,148.483
C06314=1200.594,200.235,-58.111,-177.650,6.450,148.482
C06315=1200.589,200.484,-58.135,-177.647,6.452,148.482
C06316=1200.585,200.733,-58.159,-177.645,6.454,148.482
C06317=1200.580,200.981,-58.183,-177.642,6.456,148.481
C06318=1200.576,201.231,-58.206,-177.640,6.458,148.481
C06319=1200.572,201.479,-58.231,-177.636,6.460,148.481
C06320=1200.566,201.728,-58.254,-177.634,6.462,148.480
C06321=1200.562,201.977,-58.279,-177.631,6.464,148.480
C06322=1200.557,202.226,-58.302,-177.628,6.466,148.480
C06323=1200.553,202.474,-58.326,-177.626,6.468,148.480
C06324=1200.548,202.723,-58.349,-177.624,6.470,148.479
C06325=1200.544,202.972,-58.373,-177.621,6.471,148.479
C06326=1200.539,203.221,-58.398,-177.618,6.473,148.479
C06327=1200.534,203.470,-58.422,-177.616,6.475,148.478
C06328=1200.530,203.719,-58.446,-177.613,6.477,148.478
C06329=1200.526,203.967,-58.470,-177.610,6.479,148.477
C06330=1200.521,204.216,-58.493,-177.608,6.481,148.477
C06331=1200.516,204.465,-58.518,-177.605,6.482,148.477
C06332=1200.512,204.714,-58.542,-177.603,6.484,148.477
C06333=1200.507,204.963,-58.566,-177.600,6.486,148.476
C06334=1200.503,205.211,-58.590,-177.597,6.488,148.476
C06335=1200.498,205.460,-58.615,-177.595,6.490,148.476
C06336=1200.493,205.708,-58.639,-177.592,6.492,148.475
C06337=1200.489,205.957,-58.662,-177.590,6.494,148.475
C06338=1200.485,206.207,-58.686,-177.587,6.495,148.475
C06339=1200.480,206.455,-58.711,-177.584,6.497,148.474
C06340=1200.475,206.704,-58.735,-177.582,6.500,148.474
C06341=1200.471,206.953,-58.759,-177.579,6.502,148.474
C06342=1200.466,207.201,-58.783,-177.576,6.504,148.474
C06343=1200.462,207.451,-58.808,-177.574,6.506,148.473
C06344=1200.457,207.699,-58.832,-177.571,6.507,148.473
C06345=1200.452,207.948,-58.856,-177.568,6.509,148.473
C06346=1200.447,208.197,-58.880,-177.566,6.511,148.472
C06347=1200.444,208.446,-58.904,-177.563,6.513,148.472
C06348=1200.439,208.695,-58.929,-177.561,6.515,148.472
C06349=1200.434,208.943,-58.953,-177.558,6.517,148.471
C06350=1200.429,209.192,-58.978,-177.556,6.519,148.471
C06351=1200.425,209.441,-59.002,-177.553,6.521,148.471
C06352=1200.421,209.689,-59.026,-177.550,6.522,148.470
C06353=1200.416,209.938,-59.051,-177.547,6.525,148.470
C06354=1200.411,210.186,-59.075,-177.545,6.527,148.470
C06355=1200.407,210.436,-59.100,-177.542,6.529,148.470
C06356=1200.402,210.706,-59.125,-177.540,6.531,148.469
C06357=1200.397,210.976,-59.152,-177.537,6.533,148.469
C06358=1200.392,211.247,-59.179,-177.534,6.535,148.469
C06359=1200.387,211.518,-59.206,-177.531,6.537,148.468
C06360=1200.383,211.766,-59.230,-177.528,6.539,148.468
C06361=1200.378,212.015,-59.255,-177.526,6.541,148.468
C06362=1200.373,212.263,-59.279,-177.523,6.543,148.467
C06363=1200.369,212.513,-59.304,-177.520,6.545,148.467
C06364=1200.364,212.761,-59.328,-177.518,6.547,148.467
C06365=1200.359,213.010,-59.352,-177.515,6.549,148.467
C06366=1200.355,213.259,-59.377,-177.512,6.551,148.466
C06367=1200.350,213.507,-59.401,-177.510,6.553,148.466
C06368=1200.346,213.756,-59.426,-177.507,6.555,148.466
C06369=1200.341,214.005,-59.451,-177.505,6.557,148.465
C06370=1200.337,214.254,-59.475,-177.502,6.559,148.465
C06371=1200.332,214.502,-59.500,-177.499,6.561,148.465
C06372=1200.328,214.751,-59.524,-177.496,6.563,148.464
C06373=1200.323,215.000,-59.549,-177.494,6.565,148.464
C06374=1200.319,215.249,-59.574,-177.492,6.567,148.464
C06375=1200.314,215.498,-59.598,-177.489,6.569,148.464
C06376=1200.309,215.746,-59.623,-177.486,6.571,148.463
C06377=1200.306,215.995,-59.648,-177.484,6.573,148.463
C06378=1200.301,216.243,-59.673,-177.481,6.575,148.463
C06379=1200.296,216.492,-59.697,-177.478,6.577,148.462
C06380=1200.292,216.741,-59.722,-177.476,6.579,148.462
C06381=1200.287,216.990,-59.747,-177.473,6.581,148.462
C06382=1200.283,217.238,-59.772,-177.470,6.583,148.462
C06383=1200.278,217.487,-59.796,-177.468,6.585,148.461
C06384=1200.273,217.736,-59.821,-177.466,6.587,148.461
C06385=1200.269,217.984,-59.846,-177.463,6.589,148.461
C06386=1200.264,218.233,-59.871,-177.460,6.591,148.460
C06387=1200.260,218.482,-59.895,-177.457,6.593,148.460
C06388=1200.256,218.730,-59.921,-177.454,6.595,148.460
C06389=1200.251,218.980,-59.946,-177.452,6.597,148.460
C06390=1200.246,219.229,-59.970,-177.450,6.599,148.459
C06391=1200.242,219.477,-59.996,-177.447,6.601,148.459
C06392=1200.237,219.726,-60.020,-177.444,6.603,148.459
C06393=1200.232,219.974,-60.045,-177.442,6.606,148.459
C06394=1200.229,220.223,-60.070,-177.439,6.608,148.458
C06395=1200.223,220.472,-60.095,-177.436,6.609,148.458
C06396=1200.219,220.720,-60.120,-177.434,6.611,148.458
C06397=1200.215,220.969,-60.145,-177.431,6.613,148.457
C06398=1200.210,221.218,-60.170,-177.429,6.615,148.457
C06399=1200.206,221.466,-60.195,-177.426,6.617,148.457
C06400=1200.201,221.716,-60.220,-177.423,6.620,148.457
C06401=1200.197,221.964,-60.245,-177.420,6.622,148.456
C06402=1200.192,222.213,-60.270,-177.418,6.624,148.456
C06403=1200.188,222.461,-60.295,-177.416,6.626,148.456
C06404=1200.183,222.711,-60.320,-177.413,6.627,148.455
C06405=1200.178,222.959,-60.346,-177.410,6.629,148.455
C06406=1200.174,223.208,-60.370,-177.408,6.632,148.455
C06407=1200.170,223.456,-60.395,-177.405,6.634,148.455
C06408=1200.165,223.705,-60.420,-177.402,6.636,148.454
C06409=1200.160,223.953,-60.446,-177.400,6.638,148.454
C06410=1200.156,224.202,-60.472,-177.398,6.640,148.454
C06411=1200.151,224.451,-60.496,-177.395,6.642,148.454
C06412=1200.147,224.699,-60.521,-177.392,6.644,148.453
C06413=1200.142,224.948,-60.546,-177.389,6.646,148.453
C06414=1200.138,225.197,-60.572,-177.387,6.648,148.453
C06415=1200.134,225.446,-60.598,-177.384,6.650,148.453
C06416=1200.129,225.695,-60.622,-177.382,6.652,148.452
C06417=1200.124,225.943,-60.648,-177.379,6.654,148.452
C06418=1200.120,226.191,-60.673,-177.376,6.657,148.452
C06419=1200.115,226.441,-60.698,-177.374,6.659,148.452
C06420=1200.111,226.689,-60.723,-177.371,6.661,148.451
C06421=1200.107,226.937,-60.749,-177.369,6.663,148.451
C06422=1200.102,227.187,-60.774,-177.366,6.664,148.451
C06423=1200.097,227.435,-60.799,-177.363,6.667,148.451
C06424=1200.093,227.684,-60.825,-177.361,6.669,148.450
C06425=1200.088,227.932,-60.851,-177.358,6.671,148.450
C06426=1200.084,228.181,-60.876,-177.355,6.673,148.450
C06427=1200.080,228.430,-60.901,-177.353,6.675,148.450
C06428=1200.075,228.678,-60.927,-177.351,6.677,148.449
C06429=1200.071,228.927,-60.952,-177.347,6.680,148.449
C06430=1200.066,229.176,-60.978,-177.345,6.682,148.449
C06431=1200.061,229.425,-61.003,-177.343,6.684,148.449
C06432=1200.057,229.673,-61.029,-177.340,6.685,148.448
C06433=1200.052,229.921,-61.054,-177.338,6.688,148.448
C06434=1200.048,230.170,-61.080,-177.335,6.690,148.448
C06435=1200.044,230.419,-61.106,-177.332,6.692,148.448
C06436=1200.039,230.667,-61.131,-177.330,6.694,148.447
C06437=1200.034,230.917,-61.156,-177.327,6.696,148.447
C06438=1200.030,231.165,-61.182,-177.325,6.698,148.447
C06439=1200.025,231.414,-61.207,-177.322,6.701,148.447
C06440=1200.021,231.662,-61.233,-177.319,6.703,148.446
C06441=1200.017,231.911,-61.259,-177.317,6.705,148.446
C06442=1200.012,232.159,-61.284,-177.314,6.707,148.446
C06443=1200.008,232.408,-61.310,-177.311,6.709,148.446
C06444=1200.003,232.657,-61.336,-177.309,6.711,148.445
C06445=1199.998,232.905,-61.361,-177.306,6.713,148.445
C06446=1199.994,233.154,-61.387,-177.304,6.715,148.445
C06447=1199.990,233.403,-61.413,-177.301,6.717,148.445
C06448=1199.985,233.652,-61.439,-177.298,6.720,148.445
C06449=1199.980,233.900,-61.464,-177.296,6.722,148.444
C06450=1199.976,234.149,-61.490,-177.293,6.724,148.444
C06451=1199.972,234.397,-61.516,-177.291,6.726,148.444
C06452=1199.967,234.646,-61.542,-177.288,6.729,148.444
C06453=1199.962,234.895,-61.567,-177.286,6.731,148.443
C06454=1199.958,235.143,-61.593,-177.283,6.733,148.443
C06455=1199.954,235.392,-61.619,-177.280,6.734,148.443
C06456=1199.949,235.640,-61.644,-177.278,6.737,148.443
C06457=1199.945,235.888,-61.671,-177.275,6.739,148.442
C06458=1199.940,236.138,-61.697,-177.272,6.741,148.442
C06459=1199.936,236.386,-61.723,-177.270,6.743,148.442
C06460=1199.931,236.658,-61.750,-177.267,6.746,148.442
C06461=1199.926,236.929,-61.779,-177.264,6.748,148.441
C06462=1199.922,237.201,-61.807,-177.262,6.751,148.441
C06463=1199.915,237.472,-61.836,-177.259,6.753,148.441
C06464=1199.912,237.720,-61.862,-177.256,6.755,148.441
C06465=1199.907,237.969,-61.888,-177.254,6.757,148.441
C06466=1199.903,238.218,-61.913,-177.251,6.759,148.440
C06467=1199.898,238.467,-61.940,-177.248,6.761,148.440
C06468=1199.894,238.715,-61.966,-177.246,6.764,148.440
C06469=1199.889,238.963,-61.992,-177.243,6.766,148.440
C06470=1199.885,239.212,-62.017,-177.241,6.768,148.439
C06471=1199.880,239.461,-62.044,-177.238,6.770,148.439
C06472=1199.876,239.710,-62.070,-177.235,6.773,148.439
C06473=1199.872,239.958,-62.096,-177.233,6.775,148.439
C06474=1199.867,240.207,-62.122,-177.230,6.777,148.438
C06475=1199.863,240.455,-62.148,-177.228,6.779,148.438
C06476=1199.858,240.704,-62.174,-177.225,6.781,148.438
C06477=1199.853,240.953,-62.201,-177.222,6.783,148.438
C06478=1199.849,241.201,-62.227,-177.220,6.786,148.438
C06479=1199.845,241.450,-62.253,-177.217,6.788,148.437
C06480=1199.840,241.699,-62.279,-177.215,6.790,148.437
C06481=1199.836,241.947,-62.305,-177.212,6.792,148.437
C06482=1199.831,242.196,-62.332,-177.210,6.794,148.437
C06483=1199.827,242.444,-62.358,-177.207,6.797,148.437
C06484=1199.823,242.693,-62.384,-177.204,6.799,148.436
C06485=1199.818,242.941,-62.411,-177.202,6.801,148.436
C06486=1199.814,243.190,-62.437,-177.199,6.803,148.436
C06487=1199.809,243.438,-62.464,-177.197,6.806,148.436
C06488=1199.805,243.687,-62.489,-177.194,6.808,148.435
C06489=1199.799,243.936,-62.515,-177.192,6.810,148.435
C06490=1199.795,244.184,-62.542,-177.189,6.813,148.435
C06491=1199.792,244.432,-62.568,-177.187,6.815,148.435
C06492=1199.787,244.681,-62.595,-177.184,6.817,148.435
C06493=1199.783,244.929,-62.621,-177.181,6.818,148.434
C06494=1199.778,245.178,-62.647,-177.179,6.821,148.434
C06495=1199.774,245.427,-62.674,-177.176,6.823,148.434
C06496=1199.769,245.676,-62.700,-177.174,6.825,148.434
C06497=1199.765,245.924,-62.727,-177.171,6.828,148.434
C06498=1199.760,246.173,-62.753,-177.168,6.830,148.434
C06499=1199.756,246.421,-62.780,-177.166,6.832,148.433
C06500=1199.751,246.670,-62.807,-177.163,6.835,148.433
C06501=1199.747,246.919,-62.832,-177.160,6.837,148.433
C06502=1199.742,247.167,-62.859,-177.158,6.839,148.433
C06503=1199.738,247.415,-62.886,-177.155,6.842,148.432
C06504=1199.734,247.664,-62.912,-177.153,6.844,148.432
C06505=1199.729,247.913,-62.939,-177.150,6.846,148.432
C06506=1199.725,248.161,-62.966,-177.148,6.848,148.432
C06507=1199.720,248.410,-62.992,-177.145,6.851,148.432
C06508=1199.716,248.658,-63.019,-177.143,6.853,148.432
C06509=1199.711,248.907,-63.046,-177.140,6.855,148.431
C06510=1199.707,249.155,-63.073,-177.138,6.858,148.431
C06511=1199.703,249.404,-63.098,-177.135,6.860,148.431
C06512=1199.698,249.653,-63.126,-177.133,6.862,148.431
C06513=1199.694,249.901,-63.152,-177.130,6.864,148.431
C06514=1199.689,250.149,-63.179,-177.127,6.867,148.430
C06515=1199.684,250.398,-63.205,-177.125,6.868,148.430
C06516=1199.680,250.647,-63.232,-177.122,6.871,148.430
C06517=1199.676,250.895,-63.259,-177.119,6.873,148.430
C06518=1199.671,251.144,-63.286,-177.117,6.875,148.430
C06519=1199.667,251.392,-63.312,-177.114,6.878,148.429
C06520=1199.663,251.640,-63.339,-177.112,6.880,148.429
C06521=1199.658,251.889,-63.366,-177.109,6.882,148.429
C06522=1199.654,252.138,-63.392,-177.107,6.885,148.429
C06523=1199.649,252.386,-63.419,-177.104,6.887,148.429
C06524=1199.644,252.635,-63.446,-177.101,6.890,148.429
C06525=1199.640,252.883,-63.473,-177.099,6.892,148.428
C06526=1199.636,253.131,-63.500,-177.096,6.894,148.428
C06527=1199.631,253.380,-63.527,-177.093,6.897,148.428
C06528=1199.627,253.629,-63.554,-177.091,6.899,148.428
C06529=1199.622,253.877,-63.582,-177.089,6.901,148.428
C06530=1199.618,254.126,-63.608,-177.086,6.904,148.427
C06531=1199.614,254.374,-63.635,-177.084,6.906,148.427
C06532=1199.609,254.623,-63.662,-177.081,6.908,148.427
C06533=1199.605,254.871,-63.689,-177.078,6.911,148.427
C06534=1199.601,255.119,-63.716,-177.076,6.913,148.427
C06535=1199.596,255.368,-63.743,-177.074,6.915,148.427
C06536=1199.591,255.616,-63.770,-177.070,6.917,148.426
C06537=1199.587,255.865,-63.797,-177.068,6.920,148.426
C06538=1199.583,256.114,-63.824,-177.065,6.922,148.426
C06539=1199.578,256.362,-63.851,-177.063,6.924,148.426
C06540=1199.574,256.611,-63.878,-177.061,6.927,148.426
C06541=1199.569,256.859,-63.905,-177.058,6.929,148.426
C06542=1199.565,257.107,-63.933,-177.055,6.931,148.425
C06543=1199.561,257.356,-63.960,-177.053,6.933,148.425
C06544=1199.556,257.605,-63.987,-177.050,6.936,148.425
C06545=1199.552,257.853,-64.014,-177.047,6.938,148.425
C06546=1199.547,258.102,-64.041,-177.045,6.941,148.425
C06547=1199.543,258.350,-64.068,-177.043,6.943,148.425
C06548=1199.538,258.598,-64.095,-177.040,6.945,148.424
C06549=1199.535,258.847,-64.123,-177.037,6.948,148.424
C06550=1199.530,259.095,-64.150,-177.035,6.950,148.424
C06551=1199.525,259.344,-64.177,-177.032,6.953,148.424
C06552=1199.521,259.592,-64.204,-177.029,6.955,148.424
C06553=1199.516,259.840,-64.232,-177.027,6.957,148.424
C06554=1199.512,260.089,-64.259,-177.024,6.960,148.424
C06555=1199.508,260.338,-64.286,-177.022,6.962,148.423
C06556=1199.503,260.586,-64.313,-177.019,6.965,148.423
C06557=1199.499,260.834,-64.341,-177.016,6.967,148.423
C06558=1199.495,261.084,-64.369,-177.014,6.969,148.423
C06559=1199.490,261.332,-64.396,-177.012,6.972,148.423
C06560=1199.486,261.580,-64.423,-177.009,6.974,148.422
C06561=1199.481,261.828,-64.450,-177.006,6.977,148.422
C06562=1199.477,262.078,-64.478,-177.004,6.979,148.422
C06563=1199.472,262.325,-64.506,-177.001,6.981,148.422
C06564=1199.468,262.598,-64.535,-176.999,6.984,148.422
C06565=1199.463,262.870,-64.566,-176.996,6.986,148.422
C06566=1199.458,263.144,-64.596,-176.993,6.989,148.422
C06567=1199.453,263.417,-64.625,-176.990,6.992,148.421
C06568=1199.449,263.665,-64.653,-176.988,6.994,148.421
C06569=1199.445,263.914,-64.681,-176.985,6.996,148.421
C06570=1199.440,264.162,-64.709,-176.982,6.999,148.421
C06571=1199.435,264.410,-64.736,-176.980,7.001,148.421
C06572=1199.431,264.659,-64.764,-176.977,7.004,148.421
C06573=1199.427,264.908,-64.791,-176.975,7.006,148.421
C06574=1199.422,265.155,-64.819,-176.972,7.009,148.420
C06575=1199.418,265.405,-64.846,-176.969,7.011,148.420
C06576=1199.414,265.652,-64.874,-176.967,7.013,148.420
C06577=1199.409,265.901,-64.901,-176.964,7.016,148.420
C06578=1199.405,266.149,-64.929,-176.962,7.018,148.420
C06579=1199.400,266.398,-64.957,-176.959,7.021,148.420
C06580=1199.396,266.646,-64.985,-176.957,7.023,148.419
C06581=1199.391,266.894,-65.013,-176.954,7.026,148.419
C06582=1199.387,267.143,-65.040,-176.952,7.028,148.419
C06583=1199.383,267.391,-65.068,-176.949,7.031,148.419
C06584=1199.378,267.640,-65.097,-176.946,7.033,148.419
C06585=1199.374,267.889,-65.124,-176.944,7.035,148.419
C06586=1199.369,268.136,-65.151,-176.941,7.038,148.419
C06587=1199.365,268.386,-65.179,-176.939,7.040,148.419
C06588=1199.361,268.633,-65.207,-176.936,7.043,148.418
C06589=1199.356,268.882,-65.235,-176.934,7.045,148.418
C06590=1199.352,269.130,-65.263,-176.931,7.048,148.418
C06591=1199.348,269.379,-65.290,-176.929,7.050,148.418
C06592=1199.344,269.627,-65.318,-176.926,7.053,148.418
C06593=1199.339,269.875,-65.347,-176.923,7.055,148.418
C06594=1199.334,270.124,-65.374,-176.921,7.058,148.418
C06595=1199.330,270.373,-65.402,-176.919,7.060,148.418
C06596=1199.326,270.620,-65.430,-176.915,7.063,148.417
C06597=1199.321,270.869,-65.458,-176.913,7.065,148.417
C06598=1199.317,271.117,-65.486,-176.911,7.068,148.417
C06599=1199.313,271.366,-65.514,-176.908,7.070,148.417
C06600=1199.308,271.615,-65.542,-176.905,7.073,148.417
C06601=1199.304,271.862,-65.570,-176.903,7.075,148.417
C06602=1199.300,272.111,-65.598,-176.901,7.077,148.417
C06603=1199.295,272.359,-65.626,-176.898,7.080,148.416
C06604=1199.291,272.608,-65.654,-176.896,7.082,148.416
C06605=1199.286,272.856,-65.682,-176.893,7.085,148.416
C06606=1199.282,273.105,-65.710,-176.890,7.087,148.416
C06607=1199.278,273.353,-65.738,-176.888,7.090,148.416
C06608=1199.274,273.602,-65.766,-176.885,7.092,148.416
C06609=1199.269,273.850,-65.795,-176.883,7.095,148.416
C06610=1199.265,274.098,-65.823,-176.880,7.097,148.416
C06611=1199.260,274.347,-65.851,-176.877,7.100,148.416
C06612=1199.256,274.595,-65.879,-176.875,7.102,148.416
C06613=1199.252,274.843,-65.907,-176.873,7.105,148.415
C06614=1199.247,275.092,-65.936,-176.870,7.107,148.415
C06615=1199.243,275.340,-65.963,-176.867,7.110,148.415
C06616=1199.238,275.589,-65.992,-176.865,7.112,148.415
C06617=1199.234,275.837,-66.020,-176.862,7.115,148.415
C06618=1199.230,276.085,-66.049,-176.860,7.117,148.415
C06619=1199.225,276.333,-66.077,-176.857,7.120,148.415
C06620=1199.221,276.582,-66.105,-176.854,7.123,148.415
C06621=1199.216,276.830,-66.133,-176.852,7.125,148.415
C06622=1199.212,277.079,-66.162,-176.849,7.128,148.414
C06623=1199.208,277.326,-66.190,-176.847,7.130,148.414
C06624=1199.204,277.575,-66.218,-176.844,7.133,148.414
C06625=1199.200,277.824,-66.247,-176.842,7.135,148.414
C06626=1199.195,278.072,-66.276,-176.839,7.138,148.414
C06627=1199.191,278.320,-66.304,-176.837,7.140,148.414
C06628=1199.186,278.569,-66.332,-176.834,7.143,148.414
C06629=1199.182,278.817,-66.360,-176.832,7.145,148.414
C06630=1199.177,279.065,-66.389,-176.829,7.148,148.413
C06631=1199.173,279.313,-66.417,-176.827,7.150,148.413
C06632=1199.169,279.562,-66.446,-176.824,7.153,148.413
C06633=1199.165,279.810,-66.474,-176.822,7.156,148.413
C06634=1199.160,280.059,-66.503,-176.819,7.159,148.413
C06635=1199.155,280.307,-66.532,-176.816,7.160,148.413
C06636=1199.152,280.555,-66.560,-176.814,7.163,148.413
C06637=1199.147,280.804,-66.589,-176.811,7.166,148.413
C06638=1199.143,281.051,-66.617,-176.809,7.169,148.413
C06639=1199.139,281.300,-66.646,-176.806,7.172,148.413
C06640=1199.134,281.549,-66.675,-176.804,7.173,148.413
C06641=1199.130,281.797,-66.702,-176.801,7.177,148.412
C06642=1199.126,282.045,-66.732,-176.799,7.179,148.412
C06643=1199.120,282.293,-66.760,-176.796,7.182,148.412
C06644=1199.117,282.541,-66.789,-176.794,7.184,148.412
C06645=1199.113,282.790,-66.818,-176.791,7.187,148.412
C06646=1199.107,283.038,-66.846,-176.789,7.189,148.412
C06647=1199.104,283.286,-66.875,-176.786,7.192,148.412
C06648=1199.100,283.535,-66.904,-176.783,7.195,148.412
C06649=1199.095,283.783,-66.933,-176.781,7.197,148.412
C06650=1199.091,284.031,-66.961,-176.778,7.200,148.412
C06651=1199.086,284.280,-66.990,-176.776,7.202,148.412
C06652=1199.082,284.528,-67.019,-176.773,7.205,148.411
C06653=1199.077,284.777,-67.048,-176.771,7.207,148.411
C06654=1199.074,285.025,-67.076,-176.768,7.210,148.411
C06655=1199.069,285.274,-67.105,-176.765,7.213,148.411
C06656=1199.065,285.521,-67.134,-176.763,7.215,148.411
C06657=1199.060,285.770,-67.163,-176.761,7.218,148.411
C06658=1199.057,286.018,-67.192,-176.758,7.220,148.411
C06659=1199.051,286.266,-67.220,-176.755,7.223,148.411
C06660=1199.047,286.514,-67.250,-176.753,7.225,148.411
C06661=1199.043,286.763,-67.279,-176.750,7.228,148.411
C06662=1199.039,287.012,-67.308,-176.748,7.231,148.411
C06663=1199.035,287.259,-67.336,-176.746,7.234,148.411
C06664=1199.030,287.508,-67.365,-176.743,7.237,148.411
C06665=1199.026,287.756,-67.395,-176.740,7.238,148.410
C06666=1199.022,288.004,-67.424,-176.738,7.241,148.410
C06667=1199.017,288.252,-67.452,-176.735,7.244,148.410
C06668=1199.013,288.527,-67.485,-176.733,7.247,148.410
C06669=1199.008,288.801,-67.517,-176.730,7.250,148.410
C06670=1199.002,289.076,-67.549,-176.727,7.253,148.410
C06671=1198.998,289.350,-67.581,-176.724,7.255,148.410
C06672=1198.993,289.599,-67.610,-176.721,7.258,148.410
C06673=1198.989,289.847,-67.640,-176.719,7.261,148.410
C06674=1198.985,290.095,-67.669,-176.717,7.264,148.410
C06675=1198.981,290.343,-67.697,-176.714,7.267,148.410
C06676=1198.977,290.591,-67.726,-176.712,7.269,148.410
C06677=1198.972,290.840,-67.756,-176.709,7.272,148.410
C06678=1198.968,291.088,-67.785,-176.706,7.275,148.410
C06679=1198.964,291.336,-67.815,-176.704,7.277,148.410
C06680=1198.959,291.585,-67.843,-176.702,7.280,148.410
C06681=1198.955,291.833,-67.872,-176.699,7.282,148.409
C06682=1198.951,292.081,-67.902,-176.696,7.285,148.409
C06683=1198.946,292.329,-67.931,-176.694,7.288,148.409
C06684=1198.942,292.577,-67.961,-176.691,7.290,148.409
C06685=1198.938,292.826,-67.990,-176.689,7.293,148.409
C06686=1198.934,293.074,-68.020,-176.687,7.295,148.409
C06687=1198.929,293.322,-68.048,-176.684,7.298,148.409
C06688=1198.925,293.570,-68.077,-176.681,7.301,148.409
C06689=1198.920,293.819,-68.107,-176.679,7.303,148.409
C06690=1198.916,294.067,-68.136,-176.676,7.306,148.409
C06691=1198.912,294.315,-68.166,-176.674,7.309,148.409
C06692=1198.908,294.563,-68.195,-176.671,7.312,148.409
C06693=1198.904,294.812,-68.225,-176.669,7.315,148.409
C06694=1198.899,295.060,-68.254,-176.667,7.317,148.409
C06695=1198.895,295.308,-68.284,-176.664,7.320,148.409
C06696=1198.890,295.556,-68.313,-176.661,7.323,148.409
C06697=1198.886,295.804,-68.343,-176.659,7.325,148.409
C06698=1198.881,296.053,-68.372,-176.656,7.328,148.409
C06699=1198.877,296.301,-68.402,-176.654,7.331,148.409
C06700=1198.873,296.549,-68.431,-176.652,7.333,148.409
C06701=1198.869,296.797,-68.461,-176.649,7.336,148.409
C06702=1198.865,297.046,-68.490,-176.646,7.339,148.409
C06703=1198.861,297.293,-68.520,-176.644,7.342,148.409
C06704=1198.857,297.542,-68.550,-176.641,7.345,148.409
C06705=1198.852,297.790,-68.580,-176.639,7.347,148.408
C06706=1198.848,298.038,-68.609,-176.636,7.350,148.408
C06707=1198.843,298.287,-68.639,-176.634,7.353,148.408
C06708=1198.839,298.535,-68.668,-176.632,7.355,148.408
C06709=1198.835,298.783,-68.698,-176.629,7.358,148.408
C06710=1198.831,299.031,-68.728,-176.626,7.361,148.408
C06711=1198.826,299.279,-68.758,-176.624,7.363,148.408
C06712=1198.822,299.528,-68.787,-176.621,7.366,148.408
C06713=1198.818,299.776,-68.817,-176.619,7.369,148.408
C06714=1198.814,300.024,-68.846,-176.617,7.371,148.408
C06715=1198.809,300.272,-68.877,-176.614,7.374,148.408
C06716=1198.805,300.521,-68.906,-176.611,7.377,148.408
C06717=1198.801,300.769,-68.936,-176.609,7.380,148.408
C06718=1198.796,301.017,-68.965,-176.606,7.383,148.408
C06719=1198.792,301.265,-68.996,-176.604,7.386,148.408
C06720=1198.788,301.513,-69.025,-176.602,7.388,148.408
C06721=1198.783,301.762,-69.055,-176.599,7.391,148.408
C06722=1198.780,302.009,-69.085,-176.597,7.393,148.408
C06723=1198.775,302.258,-69.115,-176.594,7.396,148.408
C06724=1198.771,302.506,-69.145,-176.591,7.399,148.408
C06725=1198.767,302.754,-69.175,-176.589,7.401,148.408
C06726=1198.762,303.002,-69.205,-176.586,7.404,148.408
C06727=1198.758,303.250,-69.235,-176.584,7.407,148.408
C06728=1198.754,303.498,-69.264,-176.582,7.409,148.408
C06729=1198.749,303.747,-69.294,-176.579,7.413,148.408
C06730=1198.745,303.994,-69.325,-176.577,7.416,148.408
C06731=1198.740,304.243,-69.355,-176.575,7.418,148.408
C06732=1198.736,304.491,-69.385,-176.572,7.421,148.408
C06733=1198.732,304.739,-69.414,-176.569,7.424,148.408
C06734=1198.727,304.987,-69.445,-176.566,7.427,148.408
C06735=1198.723,305.235,-69.475,-176.564,7.429,148.408
C06736=1198.719,305.484,-69.506,-176.562,7.432,148.408
C06737=1198.715,305.732,-69.535,-176.559,7.435,148.408
C06738=1198.711,305.980,-69.565,-176.557,7.437,148.408
C06739=1198.706,306.228,-69.595,-176.555,7.441,148.408
C06740=1198.702,306.476,-69.625,-176.552,7.444,148.408
C06741=1198.697,306.724,-69.656,-176.550,7.446,148.408
C06742=1198.693,306.972,-69.686,-176.547,7.449,148.408
C06743=1198.689,307.220,-69.716,-176.544,7.452,148.408
C06744=1198.685,307.469,-69.746,-176.542,7.454,148.408
C06745=1198.681,307.717,-69.777,-176.540,7.457,148.408
C06746=1198.676,307.965,-69.807,-176.537,7.460,148.408
C06747=1198.672,308.213,-69.837,-176.535,7.463,148.408
C06748=1198.668,308.461,-69.867,-176.532,7.466,148.408
C06749=1198.663,308.709,-69.897,-176.530,7.469,148.408
C06750=1198.659,308.957,-69.928,-176.528,7.471,148.408
C06751=1198.655,309.206,-69.959,-176.525,7.474,148.408
C06752=1198.651,309.453,-69.989,-176.522,7.477,148.408
C06753=1198.646,309.702,-70.019,-176.521,7.480,148.408
C06754=1198.642,309.950,-70.049,-176.518,7.483,148.408
C06755=1198.638,310.198,-70.080,-176.515,7.486,148.408
C06756=1198.634,310.446,-70.109,-176.512,7.489,148.408
C06757=1198.630,310.695,-70.141,-176.510,7.491,148.408
C06758=1198.625,310.942,-70.171,-176.508,7.494,148.408
C06759=1198.621,311.190,-70.201,-176.505,7.497,148.408
C06760=1198.617,311.438,-70.232,-176.503,7.499,148.408
C06761=1198.613,311.687,-70.262,-176.501,7.502,148.408
C06762=1198.608,311.935,-70.293,-176.498,7.505,148.408
C06763=1198.604,312.183,-70.324,-176.496,7.508,148.408
C06764=1198.600,312.431,-70.354,-176.494,7.511,148.408
C06765=1198.595,312.679,-70.384,-176.491,7.514,148.408
C06766=1198.591,312.927,-70.416,-176.488,7.517,148.408
C06767=1198.587,313.175,-70.446,-176.486,7.519,148.408
C06768=1198.583,313.423,-70.477,-176.484,7.522,148.408
C06769=1198.578,313.671,-70.507,-176.481,7.525,148.408
C06770=1198.575,313.920,-70.537,-176.479,7.528,148.408
C06771=1198.570,314.168,-70.568,-176.476,7.531,148.408
C06772=1198.565,314.444,-70.602,-176.474,7.534,148.408
C06773=1198.561,314.720,-70.637,-176.471,7.537,148.408
C06774=1198.556,314.996,-70.670,-176.469,7.540,148.408
C06775=1198.551,315.272,-70.705,-176.465,7.544,148.408
C06776=1198.547,315.521,-70.736,-176.463,7.546,148.408
C06777=1198.543,315.769,-70.767,-176.461,7.549,148.409
C06778=1198.539,316.016,-70.797,-176.458,7.552,148.409
C06779=1198.535,316.265,-70.828,-176.456,7.555,148.408
C06780=1198.530,316.513,-70.859,-176.454,7.558,148.408
C06781=1198.525,316.761,-70.889,-176.451,7.561,148.409
C06782=1198.522,317.009,-70.920,-176.449,7.564,148.409
C06783=1198.518,317.257,-70.951,-176.446,7.566,148.409
C06784=1198.513,317.505,-70.981,-176.444,7.570,148.409
C06785=1198.509,317.753,-71.013,-176.442,7.573,148.409
C06786=1198.505,318.001,-71.044,-176.439,7.575,148.409
C06787=1198.501,318.249,-71.074,-176.437,7.578,148.409
C06788=1198.497,318.498,-71.105,-176.435,7.581,148.409
C06789=1198.492,318.746,-71.136,-176.432,7.584,148.409
C06790=1198.487,318.994,-71.167,-176.430,7.587,148.409
C06791=1198.484,319.242,-71.199,-176.427,7.590,148.409
C06792=1198.479,319.490,-71.229,-176.425,7.593,148.409
C06793=1198.475,319.737,-71.260,-176.423,7.596,148.409
C06794=1198.471,319.986,-71.291,-176.420,7.598,148.409
C06795=1198.467,320.233,-71.322,-176.418,7.601,148.409
C06796=1198.463,320.482,-71.353,-176.415,7.605,148.409
C06797=1198.458,320.730,-71.384,-176.413,7.607,148.409
C06798=1198.454,320.978,-71.415,-176.411,7.610,148.409
C06799=1198.450,321.226,-71.447,-176.408,7.613,148.410
C06800=1198.445,321.474,-71.478,-176.406,7.616,148.410
C06801=1198.441,321.722,-71.509,-176.404,7.619,148.410
C06802=1198.437,321.970,-71.540,-176.401,7.622,148.410
C06803=1198.434,322.218,-71.571,-176.399,7.625,148.410
C06804=1198.429,322.466,-71.601,-176.396,7.628,148.410
C06805=1198.425,322.713,-71.633,-176.394,7.630,148.410
C06806=1198.421,322.962,-71.664,-176.392,7.634,148.410
C06807=1198.417,323.209,-71.696,-176.389,7.637,148.410
C06808=1198.413,323.458,-71.727,-176.387,7.639,148.410
C06809=1198.408,323.706,-71.757,-176.385,7.642,148.410
C06810=1198.404,323.954,-71.789,-176.382,7.645,148.410
C06811=1198.400,324.202,-71.820,-176.380,7.648,148.411
C06812=1198.396,324.450,-71.852,-176.378,7.651,148.410
C06813=1198.391,324.698,-71.883,-176.376,7.654,148.411
C06814=1198.388,324.946,-71.914,-176.373,7.657,148.411
C06815=1198.383,325.194,-71.945,-176.370,7.660,148.411
C06816=1198.379,325.442,-71.977,-176.369,7.663,148.411
C06817=1198.375,325.690,-72.008,-176.366,7.666,148.411
C06818=1198.371,325.938,-72.040,-176.364,7.669,148.411
C06819=1198.366,326.186,-72.071,-176.362,7.671,148.411
C06820=1198.362,326.434,-72.103,-176.359,7.674,148.411
C06821=1198.358,326.682,-72.134,-176.357,7.677,148.411
C06822=1198.354,326.930,-72.166,-176.355,7.681,148.411
C06823=1198.349,327.178,-72.197,-176.352,7.683,148.411
C06824=1198.345,327.426,-72.228,-176.350,7.686,148.412
C06825=1198.341,327.674,-72.260,-176.347,7.689,148.412
C06826=1198.337,327.922,-72.291,-176.345,7.693,148.412
C06827=1198.333,328.170,-72.322,-176.343,7.695,148.412
C06828=1198.328,328.418,-72.355,-176.341,7.698,148.412
C06829=1198.324,328.665,-72.386,-176.338,7.701,148.412
C06830=1198.320,328.914,-72.417,-176.336,7.705,148.412
C06831=1198.316,329.161,-72.449,-176.334,7.707,148.412
C06832=1198.312,329.409,-72.481,-176.332,7.710,148.412
C06833=1198.308,329.658,-72.512,-176.329,7.713,148.413
C06834=1198.303,329.906,-72.544,-176.327,7.716,148.413
C06835=1198.299,330.154,-72.576,-176.325,7.719,148.413
C06836=1198.295,330.401,-72.607,-176.322,7.722,148.413
C06837=1198.291,330.650,-72.638,-176.320,7.725,148.413
C06838=1198.286,330.897,-72.670,-176.317,7.728,148.413
C06839=1198.282,331.145,-72.702,-176.316,7.731,148.413
C06840=1198.278,331.393,-72.734,-176.313,7.734,148.413
C06841=1198.274,331.641,-72.766,-176.311,7.737,148.413
C06842=1198.270,331.889,-72.797,-176.309,7.740,148.414
C06843=1198.265,332.137,-72.829,-176.306,7.743,148.414
C06844=1198.261,332.385,-72.861,-176.304,7.746,148.414
C06845=1198.258,332.633,-72.892,-176.302,7.749,148.414
C06846=1198.252,332.881,-72.924,-176.300,7.752,148.414
C06847=1198.249,333.129,-72.956,-176.298,7.755,148.414
C06848=1198.245,333.377,-72.988,-176.295,7.758,148.414
C06849=1198.241,333.624,-73.020,-176.293,7.761,148.414
C06850=1198.236,333.873,-73.052,-176.291,7.764,148.415
C06851=1198.232,334.120,-73.084,-176.289,7.767,148.415
C06852=1198.228,334.368,-73.115,-176.286,7.770,148.415
C06853=1198.224,334.616,-73.148,-176.284,7.773,148.415
C06854=1198.220,334.864,-73.179,-176.282,7.776,148.415
C06855=1198.216,335.112,-73.211,-176.280,7.779,148.415
C06856=1198.211,335.360,-73.244,-176.277,7.782,148.415
C06857=1198.207,335.607,-73.275,-176.275,7.786,148.416
C06858=1198.203,335.856,-73.308,-176.273,7.788,148.416
C06859=1198.199,336.104,-73.339,-176.271,7.791,148.416
C06860=1198.195,336.352,-73.371,-176.268,7.794,148.416
C06861=1198.190,336.599,-73.403,-176.266,7.798,148.416
C06862=1198.186,336.848,-73.435,-176.264,7.800,148.416
C06863=1198.182,337.096,-73.468,-176.262,7.803,148.416
C06864=1198.178,337.343,-73.499,-176.260,7.807,148.417
C06865=1198.174,337.591,-73.531,-176.257,7.810,148.417
C06866=1198.170,337.840,-73.563,-176.255,7.812,148.417
C06867=1198.166,338.088,-73.595,-176.253,7.816,148.417
C06868=1198.161,338.335,-73.628,-176.251,7.819,148.417
C06869=1198.157,338.583,-73.660,-176.249,7.822,148.417
C06870=1198.153,338.831,-73.692,-176.246,7.824,148.417
C06871=1198.149,339.078,-73.724,-176.244,7.828,148.418
C06872=1198.144,339.327,-73.756,-176.242,7.831,148.418
C06873=1198.141,339.574,-73.789,-176.240,7.834,148.418
C06874=1198.136,339.822,-73.821,-176.238,7.837,148.418
C06875=1198.133,340.071,-73.853,-176.235,7.840,148.418
C06876=1198.128,340.348,-73.889,-176.233,7.843,148.418
C06877=1198.123,340.627,-73.926,-176.231,7.847,148.419
C06878=1198.118,340.906,-73.962,-176.228,7.851,148.419
C06879=1198.113,341.184,-73.998,-176.226,7.854,148.419
C06880=1198.110,341.432,-74.030,-176.224,7.857,148.419
C06881=1198.106,341.680,-74.063,-176.222,7.860,148.419
C06882=1198.101,341.928,-74.095,-176.219,7.863,148.420
C06883=1198.097,342.175,-74.127,-176.217,7.866,148.420
C06884=1198.093,342.423,-74.160,-176.215,7.869,148.420
C06885=1198.089,342.671,-74.192,-176.213,7.872,148.420
C06886=1198.085,342.919,-74.225,-176.211,7.875,148.420
C06887=1198.080,343.167,-74.257,-176.209,7.879,148.421
C06888=1198.076,343.415,-74.289,-176.207,7.881,148.421
C06889=1198.072,343.662,-74.322,-176.205,7.885,148.421
C06890=1198.067,343.911,-74.354,-176.203,7.888,148.421
C06891=1198.064,344.158,-74.387,-176.200,7.891,148.421
C06892=1198.060,344.406,-74.419,-176.199,7.894,148.422
C06893=1198.055,344.654,-74.453,-176.196,7.897,148.422
C06894=1198.051,344.902,-74.484,-176.194,7.900,148.422
C06895=1198.047,345.150,-74.517,-176.192,7.904,148.422
C06896=1198.043,345.398,-74.550,-176.190,7.906,148.422
C06897=1198.039,345.646,-74.582,-176.188,7.909,148.422
C06898=1198.035,345.893,-74.615,-176.185,7.913,148.423
C06899=1198.031,346.141,-74.648,-176.183,7.916,148.423
C06900=1198.027,346.389,-74.680,-176.182,7.919,148.423
C06901=1198.022,346.636,-74.712,-176.179,7.922,148.423
C06902=1198.018,346.885,-74.745,-176.177,7.925,148.424
C06903=1198.014,347.132,-74.778,-176.176,7.928,148.424
C06904=1198.010,347.380,-74.810,-176.174,7.931,148.424
C06905=1198.006,347.628,-74.843,-176.171,7.935,148.424
C06906=1198.002,347.876,-74.876,-176.169,7.938,148.425
C06907=1197.997,348.124,-74.909,-176.168,7.940,148.425
C06908=1197.994,348.372,-74.941,-176.165,7.944,148.425
C06909=1197.990,348.619,-74.974,-176.163,7.947,148.425
C06910=1197.985,348.868,-75.007,-176.161,7.950,148.425
C06911=1197.980,349.115,-75.040,-176.159,7.953,148.426
C06912=1197.976,349.362,-75.073,-176.157,7.956,148.426
C06913=1197.973,349.610,-75.105,-176.155,7.960,148.426
C06914=1197.968,349.858,-75.138,-176.153,7.963,148.426
C06915=1197.964,350.106,-75.171,-176.151,7.966,148.427
C06916=1197.960,350.354,-75.204,-176.149,7.969,148.427
C06917=1197.956,350.602,-75.237,-176.147,7.972,148.427
C06918=1197.952,350.850,-75.270,-176.145,7.975,148.427
C06919=1197.948,351.097,-75.302,-176.143,7.978,148.427
C06920=1197.944,351.345,-75.335,-176.141,7.982,148.428
C06921=1197.940,351.593,-75.368,-176.139,7.985,148.428
C06922=1197.935,351.841,-75.401,-176.137,7.988,148.428
C06923=1197.931,352.089,-75.434,-176.135,7.991,148.429
C06924=1197.927,352.336,-75.467,-176.133,7.994,148.429
C06925=1197.923,352.584,-75.500,-176.132,7.997,148.429
C06926=1197.919,352.832,-75.534,-176.129,8.001,148.429
C06927=1197.915,353.080,-75.565,-176.127,8.004,148.430
C06928=1197.911,353.328,-75.599,-176.125,8.007,148.430
C06929=1197.907,353.575,-75.632,-176.124,8.010,148.430
C06930=1197.903,353.823,-75.665,-176.121,8.013,148.430
C06931=1197.899,354.071,-75.698,-176.119,8.017,148.431
C06932=1197.895,354.318,-75.731,-176.117,8.020,148.431
C06933=1197.890,354.566,-75.764,-176.116,8.023,148.431
C06934=1197.886,354.814,-75.798,-176.114,8.026,148.432
C06935=1197.882,355.062,-75.831,-176.111,8.030,148.432
C06936=1197.878,355.309,-75.864,-176.110,8.032,148.432
C06937=1197.874,355.557,-75.897,-176.108,8.036,148.432
C06938=1197.870,355.805,-75.930,-176.106,8.039,148.433
C06939=1197.866,356.053,-75.963,-176.104,8.043,148.433
C06940=1197.861,356.300,-75.996,-176.102,8.045,148.433
C06941=1197.857,356.548,-76.030,-176.100,8.048,148.433
C06942=1197.853,356.796,-76.063,-176.098,8.052,148.434
C06943=1197.849,357.043,-76.096,-176.096,8.055,148.434
C06944=1197.845,357.292,-76.129,-176.095,8.058,148.434
C06945=1197.841,357.540,-76.163,-176.092,8.062,148.435
C06946=1197.837,357.787,-76.196,-176.091,8.064,148.435
C06947=1197.833,358.035,-76.229,-176.089,8.068,148.435
C06948=1197.829,358.283,-76.262,-176.087,8.071,148.436
C06949=1197.825,358.530,-76.296,-176.085,8.075,148.436
C06950=1197.821,358.778,-76.329,-176.083,8.077,148.436
C06951=1197.817,359.025,-76.362,-176.082,8.081,148.437
C06952=1197.812,359.273,-76.396,-176.079,8.084,148.437
C06953=1197.808,359.521,-76.429,-176.078,8.087,148.437
C06954=1197.804,359.770,-76.463,-176.076,8.090,148.437
C06955=1197.800,360.017,-76.497,-176.074,8.094,148.438
C06956=1197.796,360.264,-76.530,-176.072,8.096,148.438
C06957=1197.792,360.512,-76.563,-176.071,8.100,148.438
C06958=1197.788,360.760,-76.596,-176.068,8.103,148.439
C06959=1197.784,361.007,-76.630,-176.067,8.106,148.439
C06960=1197.780,361.255,-76.663,-176.065,8.110,148.440
C06961=1197.775,361.503,-76.697,-176.063,8.113,148.440
C06962=1197.772,361.751,-76.730,-176.062,8.116,148.440
C06963=1197.768,361.998,-76.764,-176.060,8.120,148.441
C06964=1197.764,362.246,-76.797,-176.059,8.122,148.441
C06965=1197.759,362.494,-76.831,-176.057,8.126,148.441
C06966=1197.756,362.741,-76.864,-176.055,8.129,148.442
C06967=1197.751,362.989,-76.898,-176.053,8.132,148.442
C06968=1197.747,363.237,-76.932,-176.052,8.136,148.442
C06969=1197.743,363.484,-76.966,-176.050,8.139,148.443
C06970=1197.739,363.732,-76.999,-176.048,8.142,148.443
C06971=1197.735,363.980,-77.032,-176.046,8.145,148.443
C06972=1197.731,364.227,-77.066,-176.045,8.148,148.444
C06973=1197.727,364.476,-77.100,-176.043,8.152,148.444
C06974=1197.723,364.723,-77.134,-176.042,8.154,148.444
C06975=1197.719,364.971,-77.167,-176.040,8.158,148.445
C06976=1197.714,365.219,-77.201,-176.038,8.162,148.445
C06977=1197.711,365.466,-77.235,-176.037,8.164,148.446
C06978=1197.707,365.714,-77.268,-176.035,8.168,148.446
C06979=1197.703,365.961,-77.302,-176.033,8.170,148.446
C06980=1197.698,366.242,-77.340,-176.032,8.174,148.447
C06981=1197.693,366.523,-77.378,-176.030,8.178,148.447
C06982=1197.688,366.804,-77.417,-176.028,8.181,148.448
C06983=1197.684,367.085,-77.456,-176.026,8.185,148.448
C06984=1197.680,367.333,-77.489,-176.024,8.189,148.448
C06985=1197.676,367.580,-77.523,-176.023,8.191,148.449
C06986=1197.672,367.827,-77.557,-176.021,8.195,148.449
C06987=1197.668,368.076,-77.591,-176.020,8.198,148.450
C06988=1197.664,368.323,-77.624,-176.018,8.202,148.450
C06989=1197.660,368.571,-77.658,-176.017,8.204,148.450
C06990=1197.656,368.818,-77.692,-176.015,8.208,148.451
C06991=1197.651,369.067,-77.726,-176.014,8.211,148.451
C06992=1197.648,369.314,-77.760,-176.012,8.214,148.452
C06993=1197.644,369.561,-77.794,-176.011,8.217,148.452
C06994=1197.639,369.809,-77.828,-176.010,8.220,148.452
C06995=1197.636,370.057,-77.862,-176.008,8.224,148.453
C06996=1197.631,370.304,-77.896,-176.007,8.226,148.453
C06997=1197.627,370.552,-77.929,-176.005,8.230,148.454
C06998=1197.624,370.800,-77.964,-176.004,8.233,148.454
C06999=1197.619,371.047,-77.998,-176.002,8.237,148.455
C07000=1197.615,371.295,-78.031,-176.001,8.239,148.455
C07001=1197.610,371.542,-78.066,-176.000,8.242,148.455
C07002=1197.607,371.790,-78.100,-175.998,8.246,148.456
C07003=1197.603,372.038,-78.133,-175.997,8.249,148.456
C07004=1197.599,372.285,-78.168,-175.996,8.252,148.457
C07005=1197.595,372.533,-78.202,-175.994,8.255,148.457
C07006=1197.591,372.781,-78.236,-175.993,8.258,148.458
C07007=1197.587,373.028,-78.270,-175.992,8.261,148.458
C07008=1197.583,373.276,-78.304,-175.990,8.265,148.459
C07009=1197.579,373.524,-78.338,-175.989,8.268,148.459
C07010=1197.574,373.771,-78.373,-175.988,8.270,148.459
C07011=1197.571,374.019,-78.407,-175.986,8.274,148.460
C07012=1197.566,374.267,-78.441,-175.985,8.277,148.460
C07013=1197.562,374.514,-78.475,-175.984,8.280,148.461
C07014=1197.558,374.762,-78.509,-175.982,8.284,148.461
C07015=1197.554,375.009,-78.543,-175.981,8.286,148.462
C07016=1197.550,375.257,-78.578,-175.980,8.290,148.462
C07017=1197.547,375.504,-78.612,-175.979,8.292,148.463
C07018=1197.542,375.752,-78.646,-175.977,8.296,148.463
C07019=1197.539,376.000,-78.680,-175.977,8.299,148.464
C07020=1197.534,376.248,-78.714,-175.975,8.302,148.464
C07021=1197.530,376.495,-78.748,-175.974,8.305,148.464
C07022=1197.526,376.743,-78.783,-175.973,8.309,148.465
C07023=1197.522,376.990,-78.818,-175.972,8.311,148.465
C07024=1197.518,377.238,-78.852,-175.971,8.315,148.466
C07025=1197.514,377.485,-78.886,-175.970,8.317,148.466
C07026=1197.510,377.733,-78.920,-175.968,8.320,148.467
C07027=1197.506,377.981,-78.955,-175.968,8.323,148.467
C07028=1197.502,378.228,-78.989,-175.966,8.327,148.468
C07029=1197.498,378.476,-79.024,-175.965,8.330,148.468
C07030=1197.494,378.723,-79.058,-175.964,8.333,148.469
C07031=1197.490,378.970,-79.092,-175.963,8.336,148.469
C07032=1197.486,379.219,-79.127,-175.962,8.339,148.470
C07033=1197.482,379.466,-79.161,-175.961,8.342,148.470
C07034=1197.478,379.714,-79.196,-175.960,8.345,148.471
C07035=1197.473,379.961,-79.230,-175.959,8.348,148.471
C07036=1197.470,380.208,-79.264,-175.957,8.351,148.472
C07037=1197.466,380.456,-79.299,-175.956,8.354,148.472
C07038=1197.461,380.704,-79.333,-175.955,8.357,148.473
C07039=1197.458,380.952,-79.367,-175.954,8.360,148.473
C07040=1197.453,381.199,-79.402,-175.954,8.363,148.474
C07041=1197.449,381.447,-79.437,-175.952,8.366,148.474
C07042=1197.446,381.694,-79.471,-175.952,8.369,148.475
C07043=1197.441,381.942,-79.505,-175.950,8.372,148.475
C07044=1197.437,382.190,-79.540,-175.950,8.375,148.476
C07045=1197.433,382.437,-79.574,-175.949,8.378,148.477
C07046=1197.429,382.685,-79.609,-175.948,8.381,148.477
C07047=1197.425,382.932,-79.644,-175.947,8.384,148.477
C07048=1197.422,383.180,-79.678,-175.946,8.387,148.478
C07049=1197.417,383.427,-79.713,-175.945,8.390,148.478
C07050=1197.413,383.675,-79.747,-175.945,8.392,148.479
C07051=1197.409,383.923,-79.782,-175.944,8.396,148.480
C07052=1197.405,384.171,-79.816,-175.943,8.398,148.480
C07053=1197.401,384.418,-79.851,-175.942,8.401,148.481
C07054=1197.397,384.665,-79.886,-175.941,8.405,148.481
C07055=1197.393,384.913,-79.921,-175.940,8.408,148.482
C07056=1197.389,385.161,-79.955,-175.939,8.410,148.482
C07057=1197.385,385.408,-79.989,-175.938,8.414,148.483
C07058=1197.381,385.656,-80.024,-175.937,8.417,148.483
C07059=1197.376,385.903,-80.059,-175.937,8.419,148.484
C07060=1197.373,386.151,-80.093,-175.936,8.422,148.484
C07061=1197.369,386.398,-80.128,-175.935,8.425,148.485
C07062=1197.365,386.646,-80.163,-175.934,8.428,148.485
C07063=1197.360,386.893,-80.198,-175.934,8.431,148.486
C07064=1197.357,387.141,-80.232,-175.933,8.433,148.487
C07065=1197.353,387.388,-80.267,-175.932,8.436,148.487
C07066=1197.349,387.637,-80.302,-175.931,8.439,148.487
C07067=1197.344,387.883,-80.337,-175.931,8.441,148.488
C07068=1197.341,388.131,-80.371,-175.930,8.445,148.489
C07069=1197.337,388.379,-80.405,-175.930,8.448,148.489
C07070=1197.333,388.626,-80.441,-175.929,8.451,148.490
C07071=1197.328,388.873,-80.475,-175.929,8.453,148.490
C07072=1197.324,389.122,-80.510,-175.927,8.456,148.491
C07073=1197.320,389.368,-80.545,-175.927,8.459,148.491
C07074=1197.317,389.616,-80.580,-175.926,8.461,148.492
C07075=1197.312,389.864,-80.614,-175.926,8.464,148.492
C07076=1197.309,390.111,-80.650,-175.925,8.467,148.493
C07077=1197.305,390.359,-80.684,-175.925,8.470,148.494
C07078=1197.300,390.607,-80.719,-175.924,8.473,148.494
C07079=1197.297,390.854,-80.754,-175.924,8.475,148.495
C07080=1197.293,391.101,-80.788,-175.923,8.478,148.495
C07081=1197.289,391.349,-80.823,-175.922,8.481,148.496
C07082=1197.284,391.596,-80.858,-175.922,8.484,148.496
C07083=1197.280,391.844,-80.893,-175.921,8.486,148.497
C07084=1197.276,392.127,-80.933,-175.920,8.490,148.498
C07085=1197.271,392.411,-80.973,-175.920,8.492,148.498
C07086=1197.267,392.693,-81.013,-175.919,8.495,148.499
C07087=1197.262,392.976,-81.053,-175.918,8.498,148.499
C07088=1197.258,393.224,-81.088,-175.918,8.501,148.500
C07089=1197.254,393.471,-81.123,-175.917,8.504,148.500
C07090=1197.251,393.718,-81.158,-175.917,8.507,148.501
C07091=1197.247,393.967,-81.192,-175.916,8.509,148.502
C07092=1197.242,394.214,-81.227,-175.916,8.512,148.502
C07093=1197.238,394.461,-81.262,-175.915,8.514,148.503
C07094=1197.234,394.709,-81.297,-175.915,8.517,148.503
C07095=1197.230,394.956,-81.332,-175.914,8.520,148.504
C07096=1197.226,395.204,-81.367,-175.914,8.522,148.504
C07097=1197.222,395.451,-81.402,-175.913,8.525,148.505
C07098=1197.218,395.699,-81.437,-175.913,8.527,148.505
C07099=1197.214,395.946,-81.472,-175.913,8.530,148.506
C07100=1197.210,396.194,-81.507,-175.912,8.533,148.507
C07101=1197.206,396.442,-81.543,-175.912,8.535,148.507
C07102=1197.202,396.689,-81.577,-175.912,8.537,148.508
C07103=1197.199,396.936,-81.612,-175.911,8.540,148.508
C07104=1197.194,397.184,-81.647,-175.911,8.543,148.509
C07105=1197.190,397.431,-81.682,-175.910,8.545,148.509
C07106=1197.187,397.679,-81.718,-175.910,8.548,148.510
C07107=1197.182,397.926,-81.752,-175.909,8.550,148.510
C07108=1197.179,398.174,-81.788,-175.909,8.553,148.511
C07109=1197.174,398.421,-81.822,-175.908,8.556,148.511
C07110=1197.170,398.669,-81.858,-175.908,8.558,148.512
C07111=1197.166,398.917,-81.893,-175.908,8.560,148.513
C07112=1197.162,399.164,-81.928,-175.908,8.562,148.513
C07113=1197.158,399.412,-81.963,-175.907,8.566,148.514
C07114=1197.154,399.659,-81.998,-175.907,8.568,148.514
C07115=1197.150,399.906,-82.033,-175.906,8.570,148.515
C07116=1197.146,400.154,-82.068,-175.906,8.572,148.515
C07117=1197.142,400.401,-82.103,-175.905,8.575,148.516
C07118=1197.138,400.649,-82.138,-175.905,8.578,148.516
C07119=1197.134,400.897,-82.174,-175.905,8.580,148.517
C07120=1197.130,401.143,-82.209,-175.905,8.582,148.517
C07121=1197.126,401.391,-82.244,-175.904,8.584,148.518
C07122=1197.122,401.639,-82.279,-175.904,8.588,148.519
C07123=1197.118,401.886,-82.315,-175.903,8.590,148.519
C07124=1197.114,402.134,-82.349,-175.903,8.592,148.520
C07125=1197.111,402.381,-82.385,-175.903,8.594,148.520
C07126=1197.106,402.628,-82.420,-175.903,8.597,148.521
C07127=1197.102,402.876,-82.455,-175.902,8.599,148.521
C07128=1197.099,403.124,-82.491,-175.902,8.601,148.522
C07129=1197.094,403.371,-82.526,-175.902,8.603,148.522
C07130=1197.090,403.619,-82.561,-175.901,8.607,148.523
C07131=1197.087,403.866,-82.596,-175.901,8.609,148.523
C07132=1197.082,404.113,-82.631,-175.901,8.611,148.524
C07133=1197.079,404.361,-82.666,-175.900,8.613,148.524
C07134=1197.074,404.609,-82.702,-175.900,8.616,148.525
C07135=1197.070,404.856,-82.737,-175.900,8.618,148.525
C07136=1197.066,405.104,-82.772,-175.900,8.620,148.526
C07137=1197.062,405.351,-82.808,-175.900,8.622,148.527
C07138=1197.058,405.598,-82.843,-175.899,8.625,148.527
C07139=1197.054,405.846,-82.879,-175.899,8.627,148.528
C07140=1197.050,406.094,-82.913,-175.899,8.629,148.528
C07141=1197.046,406.341,-82.949,-175.899,8.632,148.529
C07142=1197.042,406.588,-82.984,-175.898,8.634,148.529
C07143=1197.038,406.836,-83.019,-175.898,8.636,148.530
C07144=1197.034,407.083,-83.054,-175.898,8.638,148.530
C07145=1197.030,407.331,-83.090,-175.898,8.641,148.531
C07146=1197.027,407.578,-83.125,-175.897,8.643,148.531
C07147=1197.022,407.825,-83.160,-175.897,8.645,148.532
C07148=1197.018,408.073,-83.196,-175.897,8.647,148.532
C07149=1197.014,408.321,-83.231,-175.897,8.650,148.533
C07150=1197.010,408.568,-83.267,-175.896,8.652,148.533
C07151=1197.006,408.815,-83.302,-175.896,8.654,148.534
C07152=1197.002,409.063,-83.337,-175.896,8.656,148.534
C07153=1196.999,409.311,-83.372,-175.896,8.659,148.535
C07154=1196.994,409.557,-83.408,-175.896,8.661,148.535
C07155=1196.991,409.805,-83.443,-175.895,8.663,148.536
C07156=1196.987,410.052,-83.479,-175.895,8.666,148.537
C07157=1196.982,410.300,-83.513,-175.895,8.668,148.537
C07158=1196.978,410.548,-83.549,-175.894,8.670,148.537
C07159=1196.974,410.795,-83.585,-175.894,8.671,148.538
C07160=1196.971,411.043,-83.620,-175.894,8.673,148.538
C07161=1196.966,411.290,-83.656,-175.894,8.676,148.539
C07162=1196.963,411.538,-83.690,-175.894,8.678,148.539
C07163=1196.959,411.785,-83.726,-175.893,8.680,148.540
C07164=1196.955,412.032,-83.761,-175.893,8.682,148.541
C07165=1196.950,412.280,-83.797,-175.893,8.685,148.541
C07166=1196.947,412.527,-83.833,-175.893,8.687,148.542
C07167=1196.943,412.775,-83.868,-175.893,8.689,148.542
C07168=1196.939,413.022,-83.904,-175.893,8.691,148.543
C07169=1196.935,413.270,-83.938,-175.893,8.693,148.543
C07170=1196.931,413.517,-83.974,-175.892,8.695,148.543
C07171=1196.927,413.765,-84.010,-175.892,8.697,148.544
C07172=1196.922,414.012,-84.045,-175.891,8.699,148.544
C07173=1196.919,414.259,-84.081,-175.891,8.702,148.545
C07174=1196.915,414.507,-84.116,-175.892,8.703,148.545
C07175=1196.911,414.754,-84.152,-175.891,8.705,148.546
C07176=1196.907,415.001,-84.187,-175.891,8.708,148.547
C07177=1196.903,415.249,-84.223,-175.891,8.710,148.547
C07178=1196.899,415.497,-84.258,-175.890,8.712,148.547
C07179=1196.895,415.745,-84.294,-175.890,8.713,148.548
C07180=1196.889,416.085,-84.343,-175.890,8.717,148.549
C07181=1196.886,416.425,-84.392,-175.890,8.719,148.549
C07182=1196.885,416.767,-84.440,-175.889,8.722,148.550
C07183=1196.888,417.106,-84.488,-175.889,8.725,148.550
C07184=1196.466,417.107,-84.527,-175.892,8.735,148.554
C07185=1196.464,416.764,-84.479,-175.893,8.733,148.554
C07186=1196.464,416.420,-84.430,-175.893,8.730,148.553
C07187=1196.468,416.077,-84.380,-175.893,8.727,148.552
C07188=1196.474,415.733,-84.331,-175.894,8.724,148.552
C07189=1196.478,415.485,-84.296,-175.893,8.723,148.551
C07190=1196.482,415.238,-84.261,-175.894,8.721,148.551
C07191=1196.485,414.991,-84.225,-175.894,8.718,148.550
C07192=1196.489,414.743,-84.190,-175.894,8.716,148.550
C07193=1196.494,414.495,-84.154,-175.895,8.714,148.549
C07194=1196.498,414.249,-84.118,-175.894,8.712,148.549
C07195=1196.501,414.001,-84.083,-175.895,8.710,148.548
C07196=1196.505,413.754,-84.047,-175.895,8.708,148.548
C07197=1196.509,413.506,-84.012,-175.895,8.706,148.547
C07198=1196.513,413.259,-83.976,-175.895,8.703,148.547
C07199=1196.518,413.011,-83.941,-175.896,8.701,148.546
C07200=1196.521,412.763,-83.906,-175.896,8.700,148.546
C07201=1196.525,412.516,-83.870,-175.896,8.698,148.545
C07202=1196.529,412.269,-83.835,-175.896,8.695,148.545
C07203=1196.533,412.022,-83.799,-175.896,8.693,148.544
C07204=1196.537,411.774,-83.764,-175.897,8.691,148.544
C07205=1196.541,411.526,-83.728,-175.897,8.689,148.543
C07206=1196.546,411.279,-83.693,-175.897,8.686,148.543
C07207=1196.549,411.031,-83.658,-175.897,8.685,148.542
C07208=1196.553,410.784,-83.622,-175.897,8.683,148.542
C07209=1196.557,410.537,-83.587,-175.897,8.680,148.541
C07210=1196.561,410.290,-83.551,-175.898,8.678,148.541
C07211=1196.565,410.042,-83.516,-175.898,8.676,148.540
C07212=1196.569,409.794,-83.481,-175.898,8.674,148.539
C07213=1196.574,409.547,-83.445,-175.898,8.671,148.539
C07214=1196.577,409.299,-83.410,-175.898,8.669,148.538
C07215=1196.581,409.052,-83.374,-175.899,8.667,148.538
C07216=1196.585,408.805,-83.339,-175.899,8.665,148.538
C07217=1196.589,408.557,-83.304,-175.900,8.663,148.537
C07218=1196.593,408.309,-83.268,-175.900,8.660,148.537
C07219=1196.596,408.062,-83.233,-175.900,8.658,148.536
C07220=1196.601,407.815,-83.198,-175.900,8.656,148.535
C07221=1196.604,407.568,-83.162,-175.901,8.653,148.535
C07222=1196.608,407.319,-83.127,-175.901,8.651,148.534
C07223=1196.613,407.072,-83.092,-175.901,8.649,148.534
C07224=1196.617,406.825,-83.056,-175.901,8.647,148.533
C07225=1196.621,406.577,-83.020,-175.902,8.644,148.533
C07226=1196.625,406.330,-82.986,-175.902,8.642,148.532
C07227=1196.629,406.082,-82.950,-175.902,8.640,148.532
C07228=1196.633,405.835,-82.915,-175.902,8.638,148.531
C07229=1196.637,405.588,-82.880,-175.902,8.635,148.531
C07230=1196.641,405.340,-82.845,-175.903,8.633,148.530
C07231=1196.644,405.093,-82.809,-175.903,8.631,148.530
C07232=1196.648,404.845,-82.774,-175.903,8.629,148.529
C07233=1196.653,404.598,-82.739,-175.903,8.626,148.529
C07234=1196.656,404.350,-82.704,-175.904,8.624,148.528
C07235=1196.660,404.103,-82.668,-175.904,8.622,148.528
C07236=1196.664,403.856,-82.633,-175.904,8.619,148.527
C07237=1196.668,403.608,-82.598,-175.904,8.617,148.526
C07238=1196.673,403.360,-82.562,-175.905,8.615,148.526
C07239=1196.677,403.113,-82.527,-175.905,8.613,148.525
C07240=1196.681,402.865,-82.492,-175.905,8.610,148.525
C07241=1196.685,402.617,-82.457,-175.906,8.607,148.524
C07242=1196.689,402.371,-82.421,-175.906,8.605,148.524
C07243=1196.693,402.123,-82.387,-175.906,8.603,148.523
C07244=1196.697,401.876,-82.351,-175.907,8.601,148.523
C07245=1196.701,401.628,-82.316,-175.907,8.598,148.522
C07246=1196.705,401.380,-82.281,-175.907,8.596,148.522
C07247=1196.709,401.133,-82.246,-175.907,8.594,148.521
C07248=1196.713,400.885,-82.211,-175.908,8.591,148.521
C07249=1196.717,400.638,-82.175,-175.908,8.588,148.520
C07250=1196.721,400.391,-82.140,-175.908,8.586,148.519
C07251=1196.725,400.143,-82.105,-175.908,8.584,148.519
C07252=1196.728,399.895,-82.070,-175.909,8.581,148.518
C07253=1196.733,399.648,-82.035,-175.909,8.578,148.518
C07254=1196.737,399.400,-82.000,-175.910,8.576,148.517
C07255=1196.740,399.153,-81.964,-175.910,8.574,148.517
C07256=1196.745,398.905,-81.930,-175.910,8.571,148.516
C07257=1196.749,398.658,-81.894,-175.911,8.568,148.515
C07258=1196.753,398.411,-81.859,-175.911,8.566,148.515
C07259=1196.757,398.163,-81.824,-175.911,8.564,148.514
C07260=1196.760,397.916,-81.789,-175.912,8.561,148.514
C07261=1196.765,397.668,-81.754,-175.912,8.558,148.513
C07262=1196.769,397.421,-81.719,-175.913,8.556,148.513
C07263=1196.773,397.172,-81.684,-175.913,8.554,148.512
C07264=1196.777,396.926,-81.649,-175.914,8.551,148.512
C07265=1196.780,396.678,-81.614,-175.914,8.548,148.511
C07266=1196.784,396.431,-81.579,-175.914,8.546,148.511
C07267=1196.788,396.183,-81.544,-175.915,8.543,148.510
C07268=1196.792,395.935,-81.509,-175.915,8.541,148.509
C07269=1196.797,395.688,-81.474,-175.916,8.538,148.509
C07270=1196.800,395.441,-81.439,-175.916,8.535,148.508
C07271=1196.805,395.193,-81.404,-175.916,8.533,148.508
C07272=1196.809,394.946,-81.369,-175.917,8.530,148.507
C07273=1196.812,394.697,-81.334,-175.917,8.528,148.507
C07274=1196.817,394.451,-81.299,-175.918,8.525,148.506
C07275=1196.821,394.203,-81.264,-175.918,8.522,148.506
C07276=1196.825,393.956,-81.229,-175.919,8.519,148.505
C07277=1196.829,393.708,-81.194,-175.919,8.517,148.504
C07278=1196.832,393.461,-81.159,-175.920,8.515,148.504
C07279=1196.836,393.213,-81.125,-175.920,8.512,148.503
C07280=1196.840,392.966,-81.089,-175.921,8.509,148.503
C07281=1196.845,392.682,-81.049,-175.921,8.506,148.502
C07282=1196.850,392.400,-81.009,-175.922,8.503,148.502
C07283=1196.854,392.116,-80.969,-175.923,8.500,148.501
C07284=1196.859,391.834,-80.930,-175.923,8.497,148.500
C07285=1196.863,391.585,-80.895,-175.924,8.494,148.500
C07286=1196.867,391.339,-80.860,-175.924,8.491,148.499
C07287=1196.871,391.090,-80.825,-175.926,8.489,148.499
C07288=1196.875,390.843,-80.790,-175.926,8.486,148.498
C07289=1196.879,390.596,-80.755,-175.927,8.483,148.498
C07290=1196.882,390.348,-80.720,-175.927,8.481,148.497
C07291=1196.887,390.101,-80.685,-175.928,8.478,148.497
C07292=1196.891,389.853,-80.650,-175.928,8.475,148.496
C07293=1196.895,389.605,-80.616,-175.929,8.472,148.495
C07294=1196.899,389.358,-80.580,-175.929,8.469,148.495
C07295=1196.903,389.111,-80.546,-175.930,8.466,148.494
C07296=1196.907,388.863,-80.512,-175.930,8.464,148.494
C07297=1196.911,388.616,-80.477,-175.931,8.461,148.493
C07298=1196.915,388.368,-80.442,-175.932,8.458,148.493
C07299=1196.919,388.120,-80.407,-175.933,8.456,148.492
C07300=1196.923,387.872,-80.372,-175.933,8.453,148.492
C07301=1196.927,387.626,-80.338,-175.934,8.450,148.491
C07302=1196.931,387.378,-80.303,-175.935,8.446,148.490
C07303=1196.935,387.130,-80.269,-175.935,8.444,148.490
C07304=1196.939,386.883,-80.233,-175.936,8.441,148.489
C07305=1196.943,386.635,-80.198,-175.937,8.438,148.489
C07306=1196.947,386.387,-80.164,-175.938,8.435,148.488
C07307=1196.951,386.139,-80.129,-175.938,8.433,148.488
C07308=1196.955,385.893,-80.094,-175.939,8.430,148.487
C07309=1196.959,385.644,-80.059,-175.940,8.427,148.487
C07310=1196.963,385.397,-80.026,-175.941,8.424,148.486
C07311=1196.967,385.149,-79.991,-175.942,8.421,148.486
C07312=1196.971,384.902,-79.956,-175.943,8.418,148.485
C07313=1196.975,384.654,-79.921,-175.943,8.415,148.484
